(* Logix 5000 project; controller PBS_Perfusion vendor 1 type 14 code 217 rev 32.14; software revision 32.03; part 11 of 27 *)
(* tags used below, declared in another part *)
   Inp_FdbkA : BOOL;   // Input Signal: Feedback A from device
   Inp_FdbkB : BOOL;   // Input Signal: Feedback B from device
   Inp_FdbkC : BOOL;   // Input Signal: Feedback C from device
   Inp_FdbkD : BOOL;   // Input Signal: Feedback D from device
   Inp_DeviceFault : BOOL;   // Input Signal: Device Fault from device
   Inp_PermOK0 : BOOL;   // 1=Permissives OK, device can be commanded to State 0
   Inp_NBPermOK0 : BOOL;   // 1=Non-Bypassable Permissives OK, device can be commanded to State 0
   Inp_PermOK1 : BOOL;   // 1=Permissives OK, device can be commanded to State 1
   Inp_NBPermOK1 : BOOL;   // 1=Non-Bypassable Permissives OK, device can be commanded to State 1
   Inp_PermOK2 : BOOL;   // 1=Permissives OK, device can be commanded to State 2
   Inp_NBPermOK2 : BOOL;   // 1=Non-Bypassable Permissives OK, device can be commanded to State 2
   Inp_PermOK3 : BOOL;   // 1=Permissives OK, device can be commanded to State 3
   Inp_NBPermOK3 : BOOL;   // 1=Non-Bypassable Permissives OK, device can be commanded to State 3
   Inp_IntlkOK : BOOL;   // 1=Interlocks OK, 0=Not OK, go to State 0
   Inp_NBIntlkOK : BOOL;   // 1=Non-Bypassable Interlocks OK, 0=Not OK, go to State 0
   Inp_IntlkAvail : BOOL;   // 1 = Interlock Availibility OK
   Inp_IOFault : BOOL;   // Input Communication Status 0=OK, 1=fail
   Inp_Sim : BOOL;   // 1=Simulate working device; 0=Control actual device
   Inp_OvrdCmd : DINT;   // Override Device Command: 0=None, 1=St.0, 2=St.1, 3=St.2, 4=St.3
   Inp_HornInh : BOOL;   // 1 = Inhibit audible alert, 0 = Alllow audible alert
   Inp_Reset : BOOL;   // 1=Reset all fault conditions and latched Alarms
   Cfg_St0onShed : BOOL;   // 1=Go to State 0 on Shed, 0=Hold position on Shed
   Cfg_NumStates : DINT;   // Number of device states (2..4)
   Cfg_FdbkSt0Check : SINT;   // Bit=1: Check Feedback in state 0, Bit=0: don't care
   Cfg_FdbkSt0State : SINT;   // (if checking) Bit=1: Feedback is 1 in State 0, Bit=0: Feedback is 0
   Cfg_FdbkSt1Check : SINT;   // Bit=1: Check Feedback in state 1, Bit=0: don't care
   Cfg_FdbkSt1State : SINT;   // (if checking) Bit=1: Feedback is 1 in State 1, Bit=0: Feedback is 0
   Cfg_FdbkSt2Check : SINT;   // Bit=1: Check Feedback in state 2, Bit=0: don't care
   Cfg_FdbkSt2State : SINT;   // (if checking) Bit=1: Feedback is 1 in State 2, Bit=0: Feedback is 0
   Cfg_FdbkSt3Check : SINT;   // Bit=1: Check Feedback in state 3, Bit=0: don't care
   Cfg_FdbkSt3State : SINT;   // (if checking) Bit=1: Feedback is 1 in State 3, Bit=0: Feedback is 0
   Cfg_HasMoreObj : BOOL;   // 1=Tells HMI an object with more info is available
   Cfg_OperSt0Prio : BOOL;   // 1=OCmd_St0 any time, 0=OCmd_St0 only when Oper selected
   Cfg_ExtSt0Prio : BOOL;   // 1=XCmd_St0 any time, 0=XCmd_St0 only when Ext selected
   Cfg_OCmdResets : BOOL;   // 1=New device OCmd resets shed latches and cleared alarms, 0=OCmdReset req'd.
   Cfg_XCmdResets : BOOL;   // 1=New device XCmd resets shed latches and cleared alarms, 0=XCmdReset req'd.
   Cfg_OvrdPermIntlk : BOOL;   // 1=Override ignores Bypassable Perm/ Intlk; 0=always use Perm/Intlk
   Cfg_ShedOnFail : BOOL;   // 1=Go to State 0 and Alarm on Fail to reach position; 0=Alarm only on Fail
   Cfg_ShedOnDeviceFault : BOOL;   // 1=Go to State 0 and Alarm on Device Fault; 0=Alarm only on Device Fault
   Cfg_ShedOnIOFault : BOOL;   // 1=Go to State 0 and Alarm on I/O Fault; 0=Alarm only on I/O Fault
   Cfg_HornOnChange : BOOL;   // 0 = Horn on energize only, 1 = Horn on any state change
   Cfg_OutAPulseT : REAL;   // Time to pulse Output A (sec) (0=output held continuously)
   Cfg_OutBPulseT : REAL;   // Time to pulse Output B (sec) (0=output held continuously)
   Cfg_OutCPulseT : REAL;   // Time to pulse Output C (sec) (0=output held continuously)
   Cfg_OutDPulseT : REAL;   // Time to pulse Output D (sec) (0=output held continuously)
   Cfg_SimFdbkT : REAL;   // Delay to echo back reaching state when in Simulation (sec)
   Cfg_StartHornT : REAL;   // Time to sound audible on commanded start (sec) (0=disabled)
   Cfg_FailT : REAL;   // Time after new state requested to reach that state before Fault (sec)
   PSet_Owner : DINT;   // Program Owner Request ID (non-zero) or Release (zero)
   PCmd_St0 : BOOL;   // Program Command to set device to State 0
   PCmd_St1 : BOOL;   // Program Command to set device to State 1
   PCmd_St2 : BOOL;   // Program Command to set device to State 2
   PCmd_St3 : BOOL;   // Program Command to set device to State 3
   PCmd_Reset : BOOL;   // Program Command to ResetShed Latches and Cleared Alarms
   PCmd_FailAck : ALIAS FOR Fail.PCmd_Ack;   // Program Command to Acknowledge Fail to Reach Target Position Alarm
   PCmd_DeviceFaultAck : ALIAS FOR DeviceFault.PCmd_Ack;   // Program Command to Acknowledge Device Fault Alarm
   PCmd_IntlkTripAck : ALIAS FOR IntlkTrip.PCmd_Ack;   // Program Command to Acknowledge Interlock Trip Alarm
   PCmd_IOFaultAck : ALIAS FOR IOFault.PCmd_Ack;   // Program Command to Acknowledge I/O Fault Alarm
   XCmd_St0 : BOOL;   // External Command to set device to State 0
   XCmd_St1 : BOOL;   // External Command to set device to State 1
   XCmd_St2 : BOOL;   // External Command to set device to State 2
   XCmd_St3 : BOOL;   // External Command to set device to State 3
   XCmd_Reset : BOOL;   // External Command to reset shed latches and cleared alarms
   Val_Cmd : DINT;   // Device Command 0=None, 1=State 0, 2=State 1, 3=State 2, 4=State 3
   Val_Owner : DINT;   // Current Object Owner ID (0=not owned)
   Sts_Available : BOOL;   // 1=Device available for control by automation (Prog)
   Sts_Bypass : BOOL;   // 1=Bypassable Interlocks and Permissives are Bypassed
   Sts_BypActive : BOOL;   // 1=Interlock / Permissive Bypassing Active (Bypassed or Maintenance)
   Sts_NotRdy : BOOL;   // 1=Device Not Ready, see detail bits for reason
   Nrdy_CfgErr : BOOL;   // 1=Device Not Ready: Configuration Error
   Nrdy_EqpFault : BOOL;   // 1=Device Not Ready: External Equipment Fault (Fault or Shed Requires Reset)
   Nrdy_Fail : BOOL;   // 1=Device Not Ready: Device Failure (Shed Requires Reset)
   Nrdy_Intlk : BOOL;   // 1=Device Not Ready: Interlock Not OK
   Nrdy_IOFault : BOOL;   // 1=Device Not Ready: I/O Fault (Shed Requires Reset)
   Nrdy_OoS : BOOL;   // 1=Device Not Ready: Device is Out of Service
   Nrdy_PrioSt0 : BOOL;   // 1=Device Not Ready: Oper/Ext Priority State 0 Command Requires Reset
   Nrdy_Perm : BOOL;   // 1=Device Not Ready: Permissive Not OK
   Sts_MaintByp : BOOL;   // 1=Device has a Maintenance Bypass function active
   Err_Timer : BOOL;   // 1=Error in Config: Feeback Check timer preset (use 0 to 2147483)
   Err_Sim : BOOL;   // 1=Error in Config: Simulation timer preset (use 0 to 2147483)
   Sts_Hand : ALIAS FOR CmdSrc.Sts_Hand;
   Sts_OoS : ALIAS FOR CmdSrc.Sts_OoS;
   Sts_Maint : ALIAS FOR CmdSrc.Sts_Maint;
   Sts_Ovrd : ALIAS FOR CmdSrc.Sts_Ovrd;
   Sts_Ext : ALIAS FOR CmdSrc.Sts_Ext;
   Sts_Prog : ALIAS FOR CmdSrc.Sts_Prog;
   Sts_Oper : ALIAS FOR CmdSrc.Sts_Oper;
   Sts_Fail : ALIAS FOR Fail.Inp;   // 1=Device failed to reach commended state
   Sts_DeviceFault : ALIAS FOR DeviceFault.Inp;   // 1=Device Fault (from Inp_DeviceFault)
   Sts_IntlkTrip : ALIAS FOR IntlkTrip.Inp;   // 1=Device commanded to State 0 by an Interlock NOT OK (one-shot)
   Sts_IOFault : ALIAS FOR IOFault.Inp;   // I/O Comm Fault Status (0=OK, 1=Bad)
   P_D4SD : BOOL;   // Unique Parameter Name for auto - discovery
   Wrk_OutDPulseT : TIMER;   // Output D Pulse Timer
   Wrk_OutCPulseT : TIMER;   // Output C Pulse Timer
   Wrk_OutBPulseT : TIMER;   // Output B Pulse Timer
   Wrk_OutAPulseT : TIMER;   // Output A Pulse Timer
   Wrk_Bypass : BOOL;   // Internal Bypassable Permissives and Interlocks are Bypassed flag
   Wrk_ActState : DINT;   // Actual State (enum)
   Fail : P_Alarm;   // Device Fail to reach commanded position
   DeviceFault : P_Alarm;   // Device Fault from device via input
   CmdSrc : P_CmdSrc;   // Control / Command Source Selection
   IOFault : P_Alarm;   // I/O Fault Alarm
   IntlkTrip : P_Alarm;   // Interlock Trip Alarm
   Wrk_ONS : SINT;   // One-Shot Store Bits
   Wrk_FdbkState : DINT;   // State(s) of device as shown by feedbacks
   Cfg_Tag : STRING_20;   // Tagname for display on HMI
   Cfg_Label : STRING_20;   // Label for graphic symbol displayed on HMI
   Cfg_Desc : STRING_40;   // Description for display on HMI
   Cfg_St3Text : STRING_8;   // Text to display in State 3
   Cfg_St2Text : STRING_8;   // Text to display in State 2
   Cfg_St1Text : STRING_8;   // Text to display in State 1
   Cfg_St0Text : STRING_8;   // Text to display in State 0
   Wrk_PermOK3 : BOOL;   // 1=Permissives are OK to go to state 3
   Wrk_PermOK2 : BOOL;   // 1=Permissives are OK to go to state 2
   Wrk_PermOK1 : BOOL;   // 1=Permissives are OK to go to state 1
   Wrk_PermOK0 : BOOL;   // 1=Permissives are OK to go to state 0
   Wrk_TgtState : DINT;   // Target device state as a number (0, 1, 2 or 3)
   Wrk_SimT : TIMER;   // Time "moving" before going to target pos. in simulation
   Wrk_FailT : TIMER;   // Failure Check timer (time to reach target position)
   Wrk_NewCmd : BOOL;   // 1=A state command has been received (even for same state)
   Wrk_PrevTgt : DINT;   // Previous Target State (last scan)
   HMI_Type : STRING_16;   // Type identifier for HMI navigation
   HMI_Lib : STRING_12;   // Display Library for Faceplate call-up
   Wrk_NotRdy : BOOL;   // Device Not Ready conditions excluding shed latches
   Wrk_NotRdy1 : BOOL;   // Device Not Ready excluding only Permissives
   Wrk_NoLongerSim : BOOL;   // Switched from Simulated to Real Device this scan
   Cfg_Area : STRING_Area;   // Process Area for security
   MRdy_Check : BOOL;   // 1=Ready for MCmd_Check, enable HMI button
   MRdy_Bypass : BOOL;   // 1=Ready for MCmd_Bypass, enable HMI button
   OCmd_ResetAckAll : BOOL;   // Oper Cmd to reset shed latches and cleared alarms, plus Acknowledge alarms
   OCmd_Reset : BOOL;   // Oper Cmd to reset shed latches and cleared alarms
   OCmd_St3 : BOOL;   // Operator Command to set device to State 3
   OCmd_St2 : BOOL;   // Operator Command to set device to State 2
   OCmd_St1 : BOOL;   // Operator Command to set device to State 1
   OCmd_St0 : BOOL;   // Operator Command to set device to State 0
   MCmd_Check : BOOL;   // Maintenance Command to Check Interlocks and Permissives
   MCmd_Bypass : BOOL;   // Maintenance Command to Bypass Interlocks and Permissives
   Wrk_StartHornT : TIMER;   // Timer for audible alert or start
   Wrk_StartHorn : BOOL;   // 1=Sound audible prior to commanded energize/ state change
   Wrk_TgtStateTmp : DINT;   // Target device state as a number (0, 1, 2 or 3) stored, before audible alert
   Wrk_AfterHornONS : BOOL;
   Wrk_AfterHornONS2 : BOOL;
   ONS : DINT[3];
   REAL : DINT;
(* P_D4SD, continued *)

ROUTINE Logic   (* ladder *)
// Normal Scan: control / monitor 2-, 3- or 4-State device
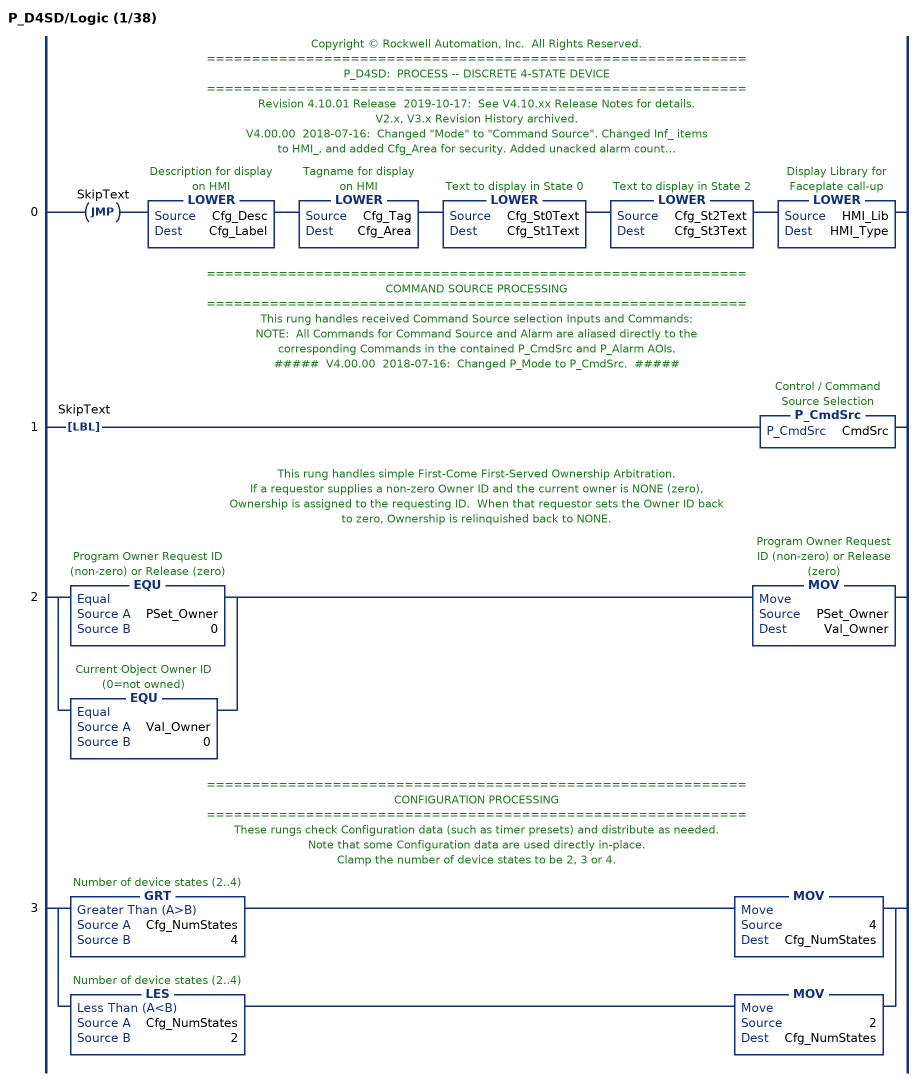
   // Copyright © Rockwell Automation, Inc.  All Rights Reserved.
   // ============================================================
   // P_D4SD:  PROCESS -- DISCRETE 4-STATE DEVICE
   // ============================================================
   // Revision 4.10.01 Release  2019-10-17:  See V4.10.xx Release Notes for details.
   // V2.x, V3.x Revision History archived.
   // V4.00.00  2018-07-16:  Changed "Mode" to "Command Source". Changed Inf_ items
   // to HMI_, and added Cfg_Area for security. Added unacked alarm count.
   // Deleted Cfg_PCmdClear; all Program Commands are now self-clearing.
   // Aligned ready bit naming with command bit names.
   // All OCmds/MCmds and ORdys/MRdys are now Local Tags.
   // Added Sts_AckReqd and Sts_ResetReqd for use by external objects.
   // Changed delay / time configuration items to REAL seconds.
   // V4.10.00  2019-03-08:  Changed availability to use input availability from interlocks.
   // Added audible alert on commanded energize/state change.
   // Added Inp_HornInh to disable Horn operation.
   // Modified logic to correct confgigurable shed action.
   // Updated to P_CmdSrc V4.10.00. Added Cfg_HasMoreObj.
   // V4.10.01  2019-10-17:  No changes, uprevved because P_CmdSrc 4.10.01 is used.
   // ============================================================
   // This Instruction controls and monitors feedback from
   // a Discrete 2-State, 3-State or 4-State Device, and provides:
   // *  Operator and Program Commands to select one of the 2, 3 or 4 states
   // *  User-configurable text labels for the states
   // *  Per-State setting, clearing or holding of four user-configurable outputs
   // *  Per-State monitoring of four feedbacks (on, off or don't care) to confirm state
   // *  Detection of failure to reach the target state (when feedbacks are used)
   // *  Monitoring of Permissive conditions to allow commanding to each state
   // *  Monitoring of Interlock conditions to return device to State 0
   // *  Simulation, providing feedback of a working device while
   //       disabling output (keeping de-energized)
   // *  Monitoring of I/O communication status
   // *  Alarms for Fail to reach target state (if feedbacks are used), Device Failure
   // (reported by device using an input), Interlock Trip, I/O Fault
   // *  "Available" status for use by automation logic to know whether
   //      the device can be controlled by other objects.
   // Command Sources are arbitrated by a P_CmdSrc Add-On Instruction instance.
   // Command Sources: Operator, Program, External, Override, Maintenance, Out of
   // Service, Hand.  Alarms are provided by P_Alarm Add-On Instruction instances.
   // ============================================================
   // SHOW LOCAL STRINGS
   // ============================================================
   // The STRINGs containing the text associated with each instance of this
   // instruction cannot be Input or Output Parameters, because STRINGs are not
   //  'atomic' types. (Inputs and Outputs must be SINT, INT, DINT, REAL, or BOOL.)
   // In order to make it easier to find and configure these STRINGs, this rung
   // was added.  THE JMP (and the LBL on the following rung)
   // MUST NOT BE REMOVED!!!
   // To view the STRINGs, go to the instruction instance (in LD or FBD), RIGHT-click
   // to bring up the context menu and select "Open Instruction Logic".
   // This rung will appear with the STRING values for the selected instance.
   // You may double-click the STRING values here to modify them as well.
   // #####  V4.00.00  2018-07-16:  Added string for Cfg_Area, renamed Inf_* to HMI_*.  #####
   0: JMP(SkipText)LOWER(Cfg_Desc,Cfg_Label)LOWER(Cfg_Tag,Cfg_Area)LOWER(Cfg_St0Text,Cfg_St1Text)LOWER(Cfg_St2Text,Cfg_St3Text)LOWER(HMI_Lib,HMI_Type);
   // ============================================================
   // COMMAND SOURCE PROCESSING
   // ============================================================
   // This rung handles received Command Source selection Inputs and Commands:
   // NOTE:  All Commands for Command Source and Alarm are aliased directly to the
   // corresponding Commands in the contained P_CmdSrc and P_Alarm AOIs.
   // #####  V4.00.00  2018-07-16:  Changed P_Mode to P_CmdSrc.  #####
   1: LBL(SkipText)P_CmdSrc(CmdSrc);
   // This rung handles simple First-Come First-Served Ownership Arbitration.
   // If a requestor supplies a non-zero Owner ID and the current owner is NONE (zero),
   // Ownership is assigned to the requesting ID.  When that requestor sets the Owner ID back
   // to zero, Ownership is relinquished back to NONE.
   2: [EQU(PSet_Owner,0) ,EQU(Val_Owner,0) ]MOV(PSet_Owner,Val_Owner);
   // ============================================================
   // CONFIGURATION PROCESSING
   // ============================================================
   // These rungs check Configuration data (such as timer presets) and distribute as needed.
   // Note that some Configuration data are used directly in-place.
   // Clamp the number of device states to be 2, 3 or 4.
   3: [GRT(Cfg_NumStates,4) MOV(4,Cfg_NumStates) ,LES(Cfg_NumStates,2) MOV(2,Cfg_NumStates) ];
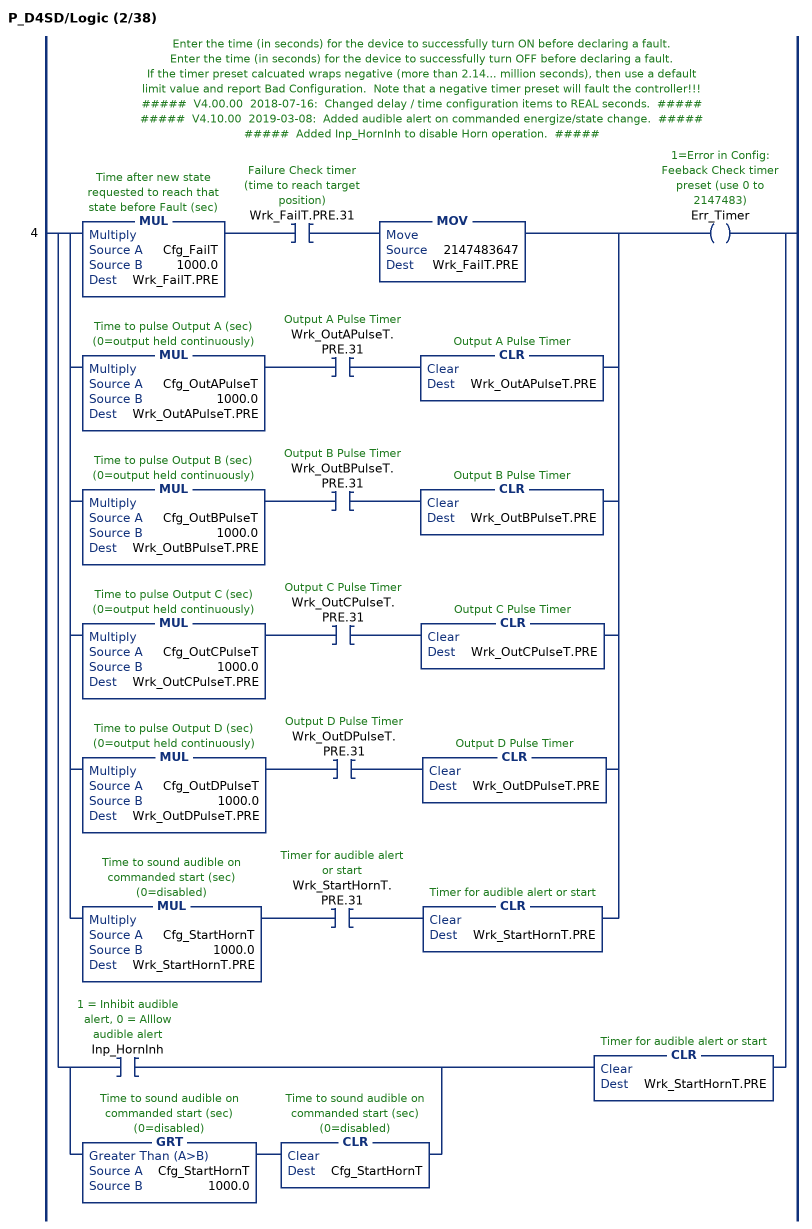
   // Enter the time (in seconds) for the device to successfully turn ON before declaring a fault.
   // Enter the time (in seconds) for the device to successfully turn OFF before declaring a fault.
   // If the timer preset calcuated wraps negative (more than 2.14... million seconds), then use a default
   // limit value and report Bad Configuration.  Note that a negative timer preset will fault the controller!!!
   // #####  V4.00.00  2018-07-16:  Changed delay / time configuration items to REAL seconds.  #####
   // #####  V4.10.00  2019-03-08:  Added audible alert on commanded energize/state change.  #####
   // #####  Added Inp_HornInh to disable Horn operation.  #####
   4: [[MUL(Cfg_FailT,1000.0,Wrk_FailT.PRE) XIC(Wrk_FailT.PRE.31) MOV(2147483647,Wrk_FailT.PRE) ,MUL(Cfg_OutAPulseT,1000.0,Wrk_OutAPulseT.PRE) XIC(Wrk_OutAPulseT.PRE.31) CLR(Wrk_OutAPulseT.PRE) ,MUL(Cfg_OutBPulseT,1000.0,Wrk_OutBPulseT.PRE) XIC(Wrk_OutBPulseT.PRE.31) CLR(Wrk_OutBPulseT.PRE) ,MUL(Cfg_OutCPulseT,1000.0,Wrk_OutCPulseT.PRE) XIC(Wrk_OutCPulseT.PRE.31) CLR(Wrk_OutCPulseT.PRE) ,MUL(Cfg_OutDPulseT,1000.0,Wrk_OutDPulseT.PRE) XIC(Wrk_OutDPulseT.PRE.31) CLR(Wrk_OutDPulseT.PRE) ,MUL(Cfg_StartHornT,1000.0,Wrk_StartHornT.PRE) XIC(Wrk_StartHornT.PRE.31) CLR(Wrk_StartHornT.PRE) ] OTE(Err_Timer) ,[XIC(Inp_HornInh) ,GRT(Cfg_StartHornT,1000.0) CLR(Cfg_StartHornT) ] CLR(Wrk_StartHornT.PRE) ];
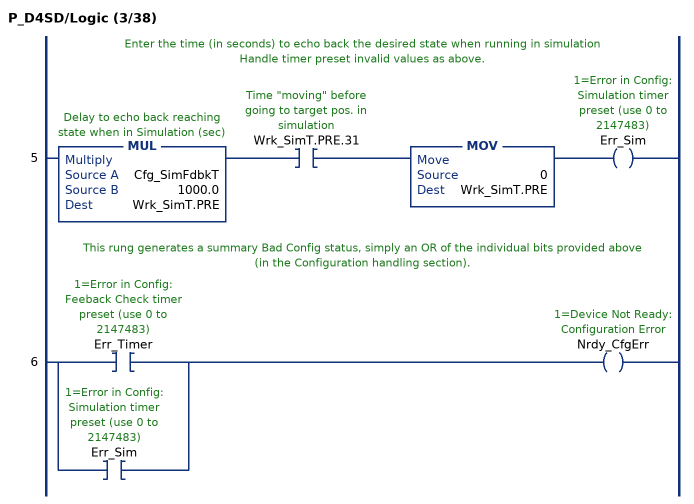
   // Enter the time (in seconds) to echo back the desired state when running in simulation
   // Handle timer preset invalid values as above.
   5: MUL(Cfg_SimFdbkT,1000.0,Wrk_SimT.PRE)XIC(Wrk_SimT.PRE.31)MOV(0,Wrk_SimT.PRE)OTE(Err_Sim);
   // This rung generates a summary Bad Config status, simply an OR of the individual bits provided above
   // (in the Configuration handling section).
   6: [XIC(Err_Timer) ,XIC(Err_Sim) ]OTE(Nrdy_CfgErr);
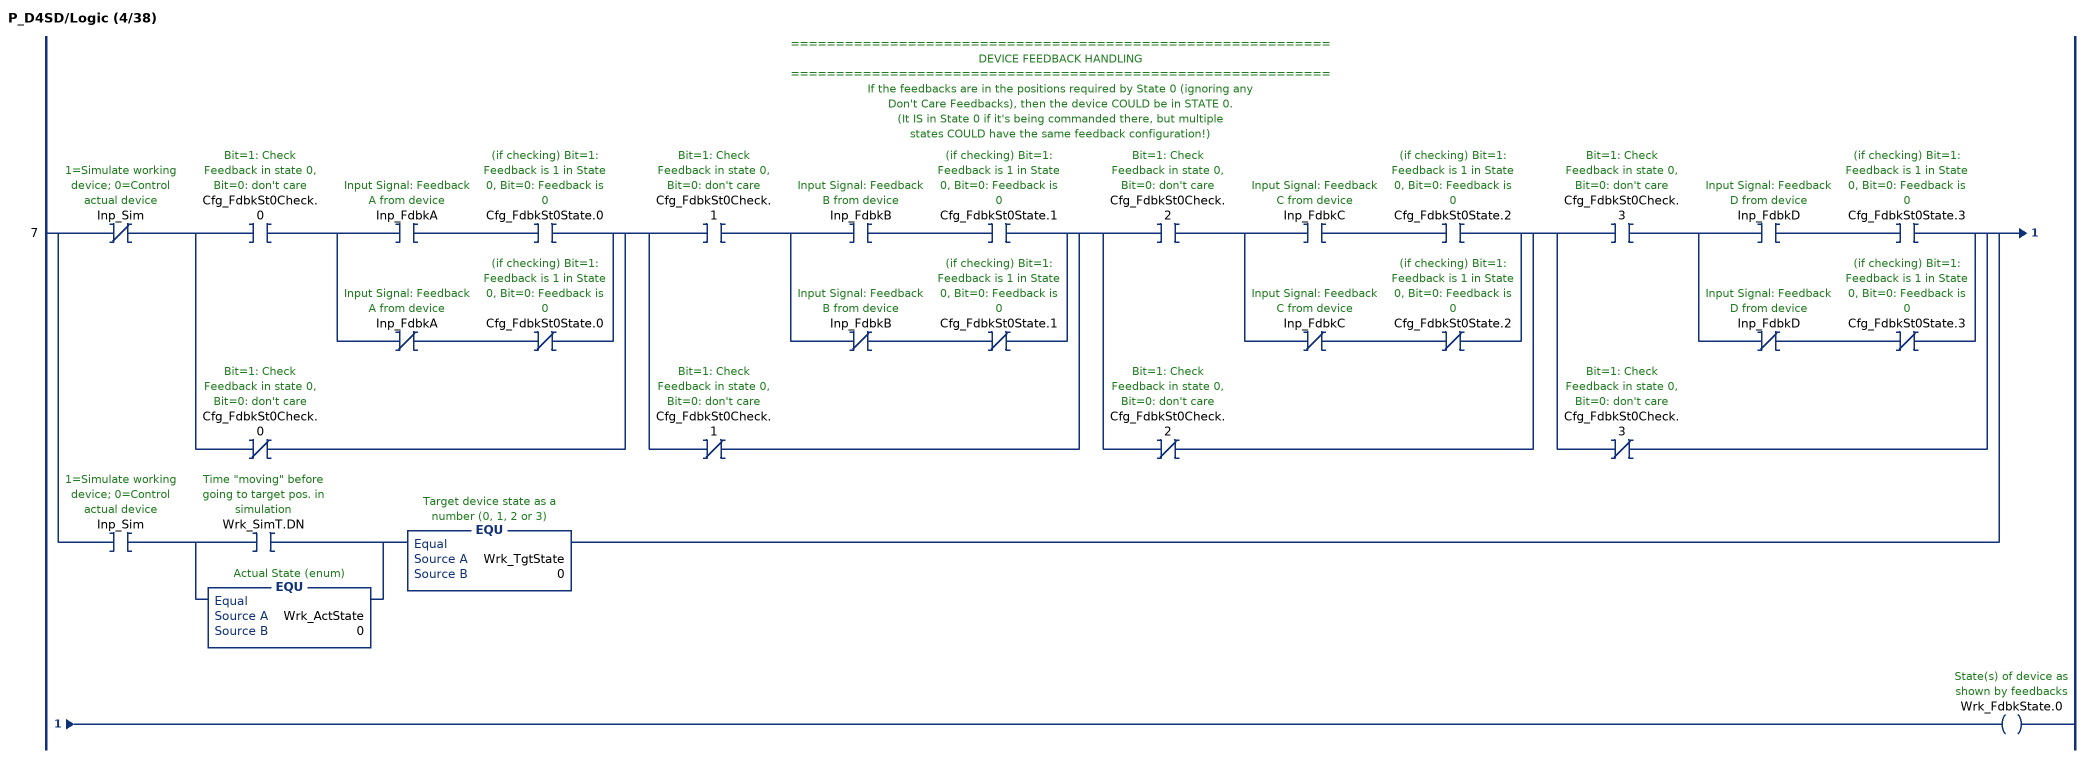
   // ============================================================
   // DEVICE FEEDBACK HANDLING
   // ============================================================
   // If the feedbacks are in the positions required by State 0 (ignoring any
   // Don't Care Feedbacks), then the device COULD be in STATE 0.
   // (It IS in State 0 if it's being commanded there, but multiple
   // states COULD have the same feedback configuration!)
   7: [XIO(Inp_Sim) [XIC(Cfg_FdbkSt0Check.0) [XIC(Inp_FdbkA) XIC(Cfg_FdbkSt0State.0) ,XIO(Inp_FdbkA) XIO(Cfg_FdbkSt0State.0) ] ,XIO(Cfg_FdbkSt0Check.0) ] [XIC(Cfg_FdbkSt0Check.1) [XIC(Inp_FdbkB) XIC(Cfg_FdbkSt0State.1) ,XIO(Inp_FdbkB) XIO(Cfg_FdbkSt0State.1) ] ,XIO(Cfg_FdbkSt0Check.1) ] [XIC(Cfg_FdbkSt0Check.2) [XIC(Inp_FdbkC) XIC(Cfg_FdbkSt0State.2) ,XIO(Inp_FdbkC) XIO(Cfg_FdbkSt0State.2) ] ,XIO(Cfg_FdbkSt0Check.2) ] [XIC(Cfg_FdbkSt0Check.3) [XIC(Inp_FdbkD) XIC(Cfg_FdbkSt0State.3) ,XIO(Inp_FdbkD) XIO(Cfg_FdbkSt0State.3) ] ,XIO(Cfg_FdbkSt0Check.3) ] ,XIC(Inp_Sim) [XIC(Wrk_SimT.DN) ,EQU(Wrk_ActState,0) ] EQU(Wrk_TgtState,0) ]OTE(Wrk_FdbkState.0);
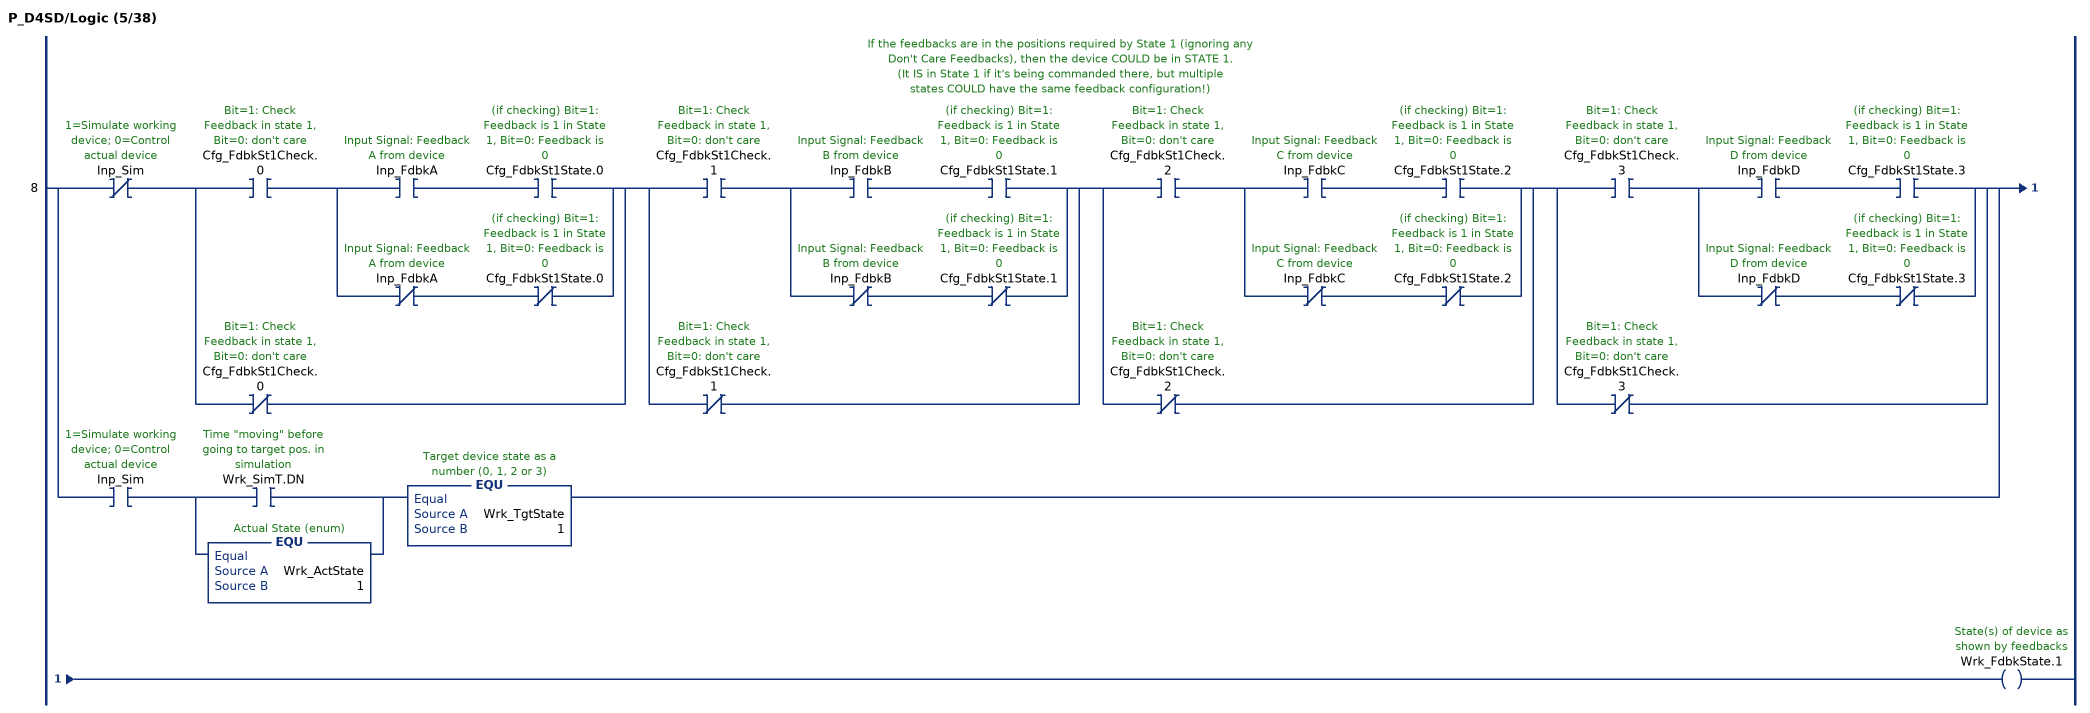
   // If the feedbacks are in the positions required by State 1 (ignoring any
   // Don't Care Feedbacks), then the device COULD be in STATE 1.
   // (It IS in State 1 if it's being commanded there, but multiple
   // states COULD have the same feedback configuration!)
   8: [XIO(Inp_Sim) [XIC(Cfg_FdbkSt1Check.0) [XIC(Inp_FdbkA) XIC(Cfg_FdbkSt1State.0) ,XIO(Inp_FdbkA) XIO(Cfg_FdbkSt1State.0) ] ,XIO(Cfg_FdbkSt1Check.0) ] [XIC(Cfg_FdbkSt1Check.1) [XIC(Inp_FdbkB) XIC(Cfg_FdbkSt1State.1) ,XIO(Inp_FdbkB) XIO(Cfg_FdbkSt1State.1) ] ,XIO(Cfg_FdbkSt1Check.1) ] [XIC(Cfg_FdbkSt1Check.2) [XIC(Inp_FdbkC) XIC(Cfg_FdbkSt1State.2) ,XIO(Inp_FdbkC) XIO(Cfg_FdbkSt1State.2) ] ,XIO(Cfg_FdbkSt1Check.2) ] [XIC(Cfg_FdbkSt1Check.3) [XIC(Inp_FdbkD) XIC(Cfg_FdbkSt1State.3) ,XIO(Inp_FdbkD) XIO(Cfg_FdbkSt1State.3) ] ,XIO(Cfg_FdbkSt1Check.3) ] ,XIC(Inp_Sim) [XIC(Wrk_SimT.DN) ,EQU(Wrk_ActState,1) ] EQU(Wrk_TgtState,1) ]OTE(Wrk_FdbkState.1);
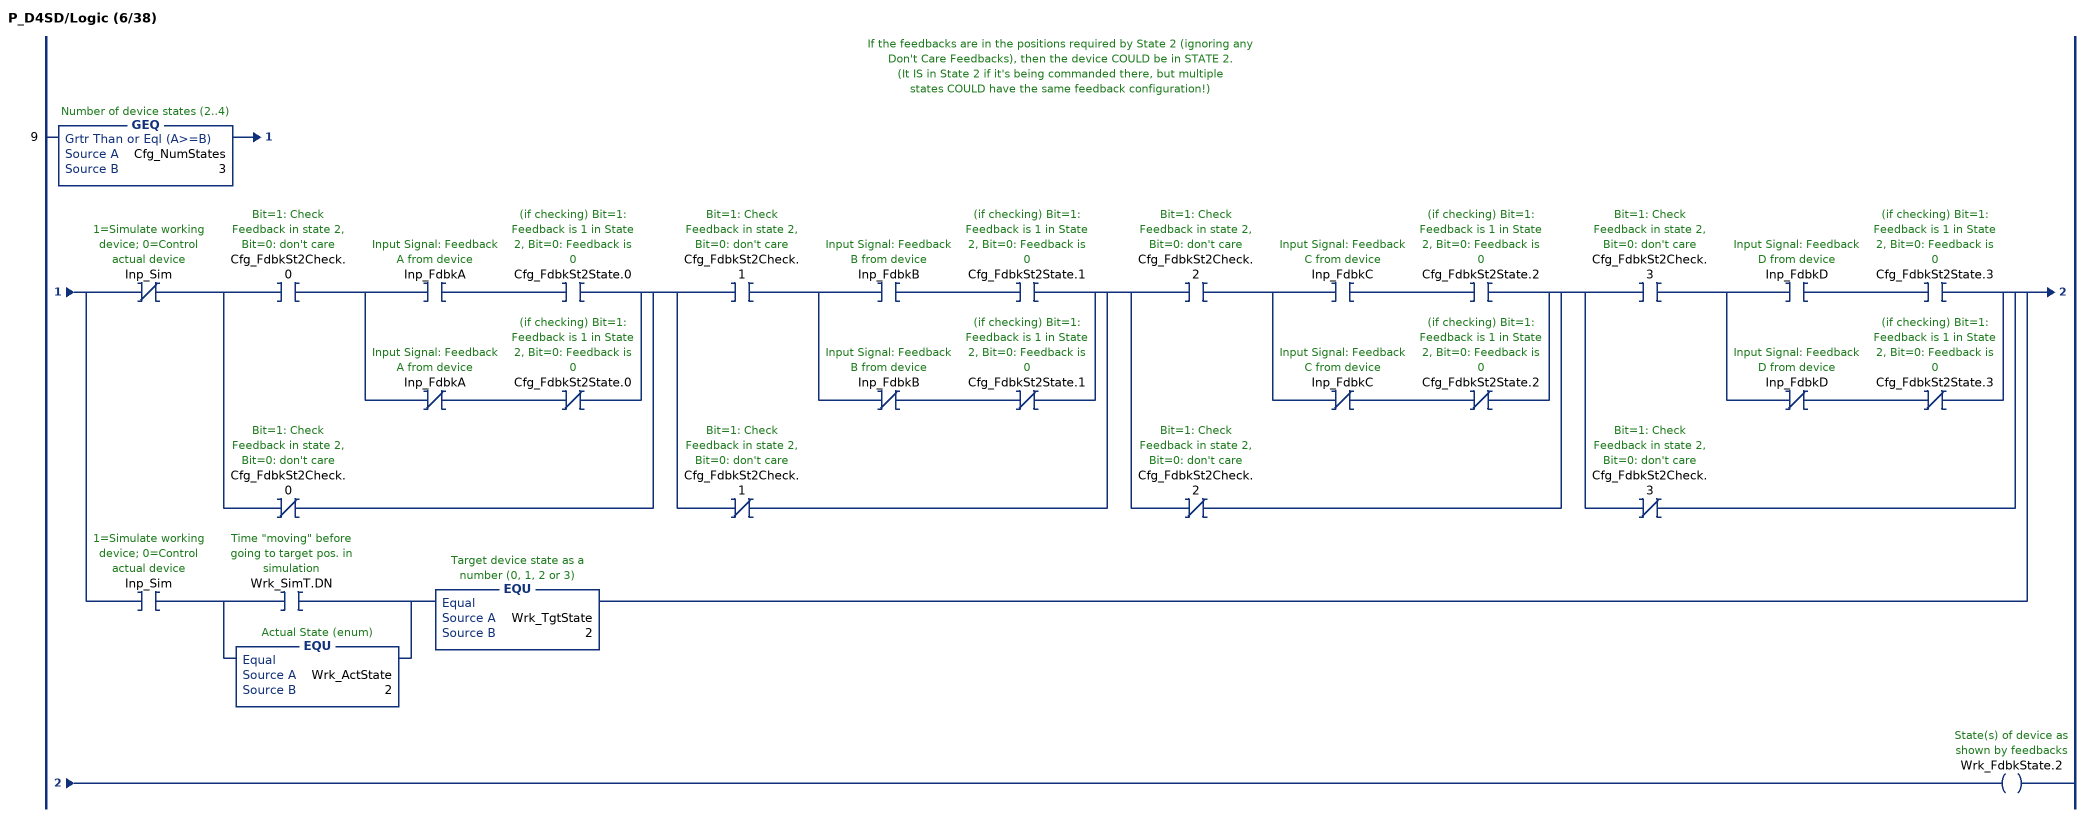
   // If the feedbacks are in the positions required by State 2 (ignoring any
   // Don't Care Feedbacks), then the device COULD be in STATE 2.
   // (It IS in State 2 if it's being commanded there, but multiple
   // states COULD have the same feedback configuration!)
   9: GEQ(Cfg_NumStates,3)[XIO(Inp_Sim) [XIC(Cfg_FdbkSt2Check.0) [XIC(Inp_FdbkA) XIC(Cfg_FdbkSt2State.0) ,XIO(Inp_FdbkA) XIO(Cfg_FdbkSt2State.0) ] ,XIO(Cfg_FdbkSt2Check.0) ] [XIC(Cfg_FdbkSt2Check.1) [XIC(Inp_FdbkB) XIC(Cfg_FdbkSt2State.1) ,XIO(Inp_FdbkB) XIO(Cfg_FdbkSt2State.1) ] ,XIO(Cfg_FdbkSt2Check.1) ] [XIC(Cfg_FdbkSt2Check.2) [XIC(Inp_FdbkC) XIC(Cfg_FdbkSt2State.2) ,XIO(Inp_FdbkC) XIO(Cfg_FdbkSt2State.2) ] ,XIO(Cfg_FdbkSt2Check.2) ] [XIC(Cfg_FdbkSt2Check.3) [XIC(Inp_FdbkD) XIC(Cfg_FdbkSt2State.3) ,XIO(Inp_FdbkD) XIO(Cfg_FdbkSt2State.3) ] ,XIO(Cfg_FdbkSt2Check.3) ] ,XIC(Inp_Sim) [XIC(Wrk_SimT.DN) ,EQU(Wrk_ActState,2) ] EQU(Wrk_TgtState,2) ]OTE(Wrk_FdbkState.2);
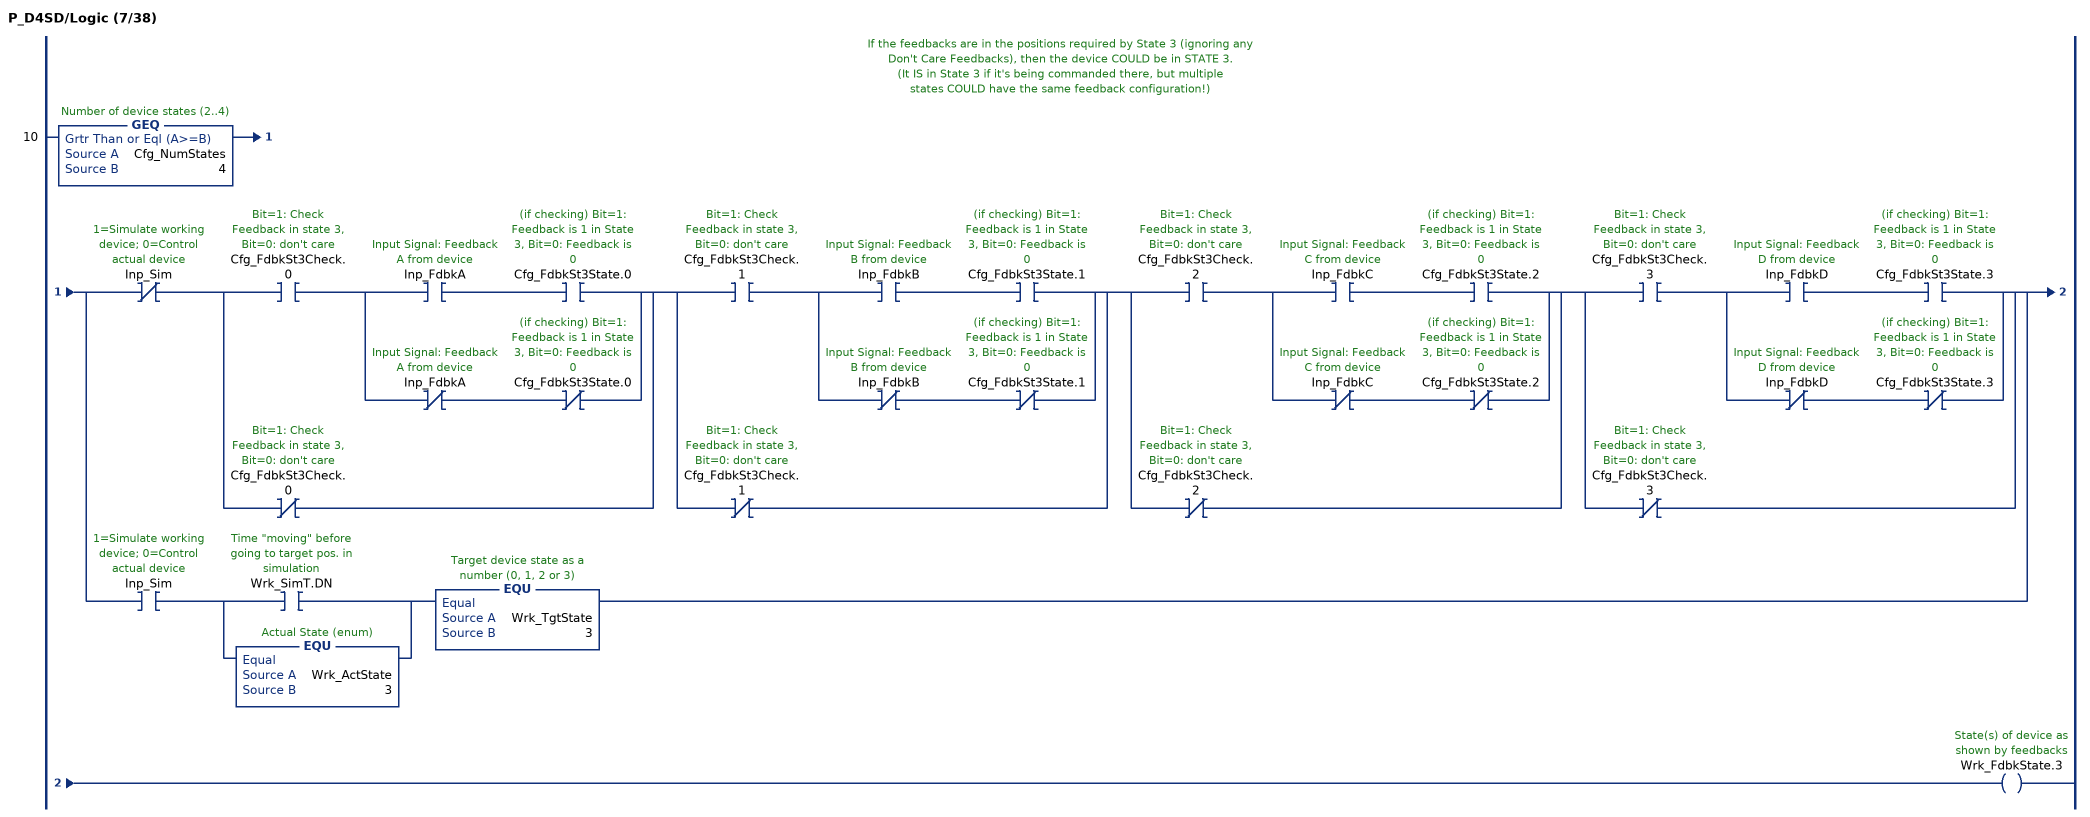
   // If the feedbacks are in the positions required by State 3 (ignoring any
   // Don't Care Feedbacks), then the device COULD be in STATE 3.
   // (It IS in State 3 if it's being commanded there, but multiple
   // states COULD have the same feedback configuration!)
   10: GEQ(Cfg_NumStates,4)[XIO(Inp_Sim) [XIC(Cfg_FdbkSt3Check.0) [XIC(Inp_FdbkA) XIC(Cfg_FdbkSt3State.0) ,XIO(Inp_FdbkA) XIO(Cfg_FdbkSt3State.0) ] ,XIO(Cfg_FdbkSt3Check.0) ] [XIC(Cfg_FdbkSt3Check.1) [XIC(Inp_FdbkB) XIC(Cfg_FdbkSt3State.1) ,XIO(Inp_FdbkB) XIO(Cfg_FdbkSt3State.1) ] ,XIO(Cfg_FdbkSt3Check.1) ] [XIC(Cfg_FdbkSt3Check.2) [XIC(Inp_FdbkC) XIC(Cfg_FdbkSt3State.2) ,XIO(Inp_FdbkC) XIO(Cfg_FdbkSt3State.2) ] ,XIO(Cfg_FdbkSt3Check.2) ] [XIC(Cfg_FdbkSt3Check.3) [XIC(Inp_FdbkD) XIC(Cfg_FdbkSt3State.3) ,XIO(Inp_FdbkD) XIO(Cfg_FdbkSt3State.3) ] ,XIO(Cfg_FdbkSt3Check.3) ] ,XIC(Inp_Sim) [XIC(Wrk_SimT.DN) ,EQU(Wrk_ActState,3) ] EQU(Wrk_TgtState,3) ]OTE(Wrk_FdbkState.3);
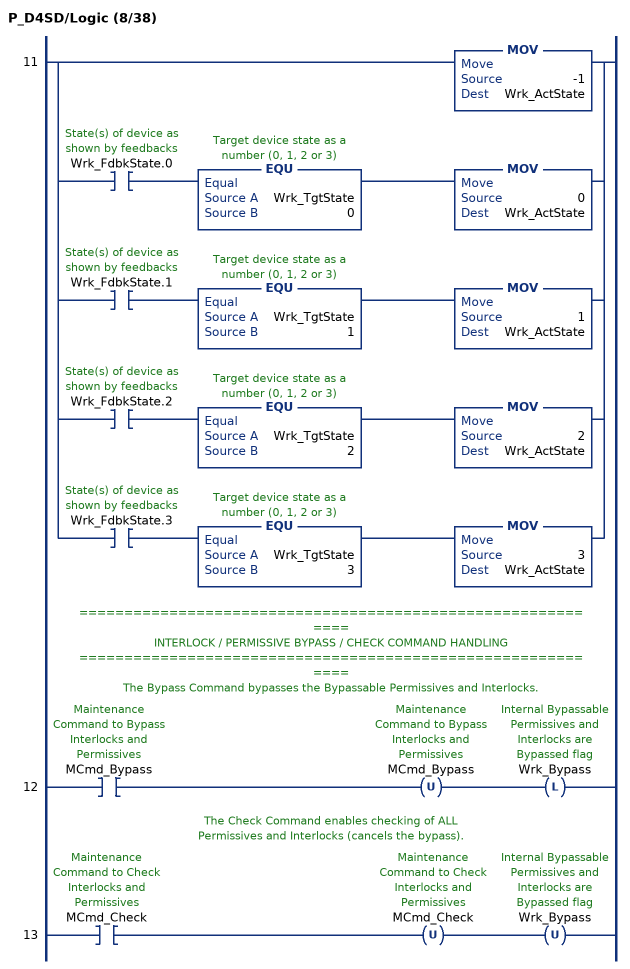
   11: [MOV(-1,Wrk_ActState) ,XIC(Wrk_FdbkState.0) EQU(Wrk_TgtState,0) MOV(0,Wrk_ActState) ,XIC(Wrk_FdbkState.1) EQU(Wrk_TgtState,1) MOV(1,Wrk_ActState) ,XIC(Wrk_FdbkState.2) EQU(Wrk_TgtState,2) MOV(2,Wrk_ActState) ,XIC(Wrk_FdbkState.3) EQU(Wrk_TgtState,3) MOV(3,Wrk_ActState) ];
   // ============================================================
   // INTERLOCK / PERMISSIVE BYPASS / CHECK COMMAND HANDLING
   // ============================================================
   // The Bypass Command bypasses the Bypassable Permissives and Interlocks.
   12: XIC(MCmd_Bypass)OTU(MCmd_Bypass)OTL(Wrk_Bypass);
   // The Check Command enables checking of ALL
   // Permissives and Interlocks (cancels the bypass).
   13: XIC(MCmd_Check)OTU(MCmd_Check)OTU(Wrk_Bypass);
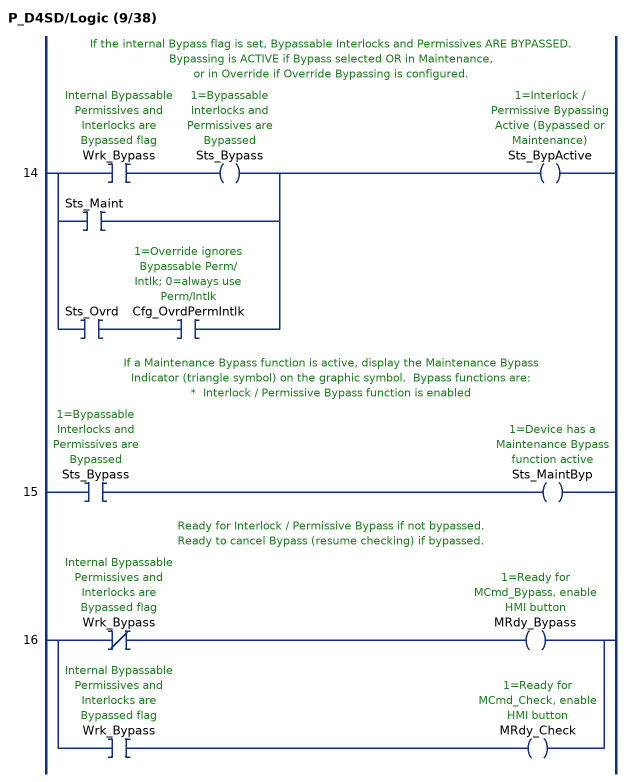
   // If the internal Bypass flag is set, Bypassable Interlocks and Permissives ARE BYPASSED.
   // Bypassing is ACTIVE if Bypass selected OR in Maintenance,
   // or in Override if Override Bypassing is configured.
   14: [XIC(Wrk_Bypass) OTE(Sts_Bypass) ,XIC(Sts_Maint) ,XIC(Sts_Ovrd) XIC(Cfg_OvrdPermIntlk) ]OTE(Sts_BypActive);
   // If a Maintenance Bypass function is active, display the Maintenance Bypass
   // Indicator (triangle symbol) on the graphic symbol.  Bypass functions are:
   // *  Interlock / Permissive Bypass function is enabled
   15: XIC(Sts_Bypass)OTE(Sts_MaintByp);
   // Ready for Interlock / Permissive Bypass if not bypassed.
   // Ready to cancel Bypass (resume checking) if bypassed.
   16: [XIO(Wrk_Bypass) OTE(MRdy_Bypass) ,XIC(Wrk_Bypass) OTE(MRdy_Check) ];
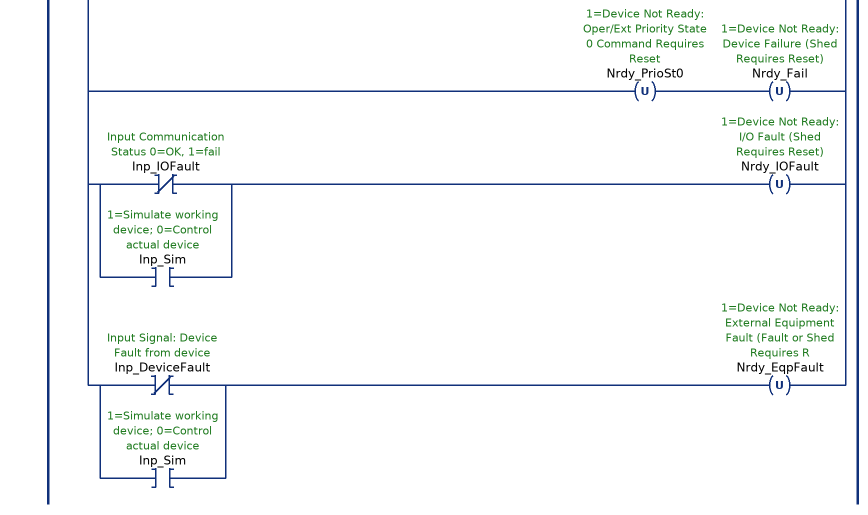
   // ============================================================
   // ALARM RESET COMMAND HANDLING
   // ============================================================
   // This rung handles the Alarm Reset Input and Commands
   // and the "Reset and Ack All" Operator Command.
   // This rung processes received Reset Commands from:
   // 1.  The Operator via HMI Operator Command, or
   // 2.  Higher-level strategies via Program Command
   // 3.  Pushbuttons or other block via Input
   // 4.  Resets initiated by other device Operator Commands (if configured to do so)
   // and forwards the Reset to ALL Alarms and latched Shed conditions.
   // #####  V4.00.00  2018-07-16:  Deleted Cfg_PCmdClear; all Program Commands are now self-clearing.  #####
   // #####  Added External Command Source and Commands.  #####
   17: [XIC(OCmd_Reset) OTU(OCmd_Reset) ,XIC(XCmd_Reset) OTU(XCmd_Reset) ,XIC(PCmd_Reset) OTU(PCmd_Reset) ,XIC(Inp_Reset) ,[XIC(OCmd_St0) XIC(Wrk_PermOK0) ,XIC(OCmd_St1) XIC(Wrk_PermOK1) ,GEQ(Cfg_NumStates,3) XIC(OCmd_St2) XIC(Wrk_PermOK2) ,GEQ(Cfg_NumStates,4) XIC(OCmd_St3) XIC(Wrk_PermOK3) ] XIC(Cfg_OCmdResets) [XIC(Sts_Oper) ,XIC(Sts_Maint) ] ,[XIC(XCmd_St0) XIC(Wrk_PermOK0) ,XIC(XCmd_St1) XIC(Wrk_PermOK1) ,GEQ(Cfg_NumStates,3) XIC(XCmd_St2) XIC(Wrk_PermOK2) ,GEQ(Cfg_NumStates,4) XIC(XCmd_St3) XIC(Wrk_PermOK3) ] XIC(Cfg_XCmdResets) XIC(Sts_Ext) ,XIC(OCmd_ResetAckAll) OTU(OCmd_ResetAckAll) [OTL(PCmd_FailAck) ,OTL(PCmd_DeviceFaultAck) ,OTL(PCmd_IntlkTripAck) ,OTL(PCmd_IOFaultAck) ] ][OTL(Fail.PCmd_Reset) OTL(DeviceFault.PCmd_Reset) ,OTL(IntlkTrip.PCmd_Reset) OTL(IOFault.PCmd_Reset) ,XIC(Sts_Fail) RES(Wrk_FailT) ,OTU(Nrdy_PrioSt0) OTU(Nrdy_Fail) ,[XIO(Inp_IOFault) ,XIC(Inp_Sim) ] OTU(Nrdy_IOFault) ,[XIO(Inp_DeviceFault) ,XIC(Inp_Sim) ] OTU(Nrdy_EqpFault) ];
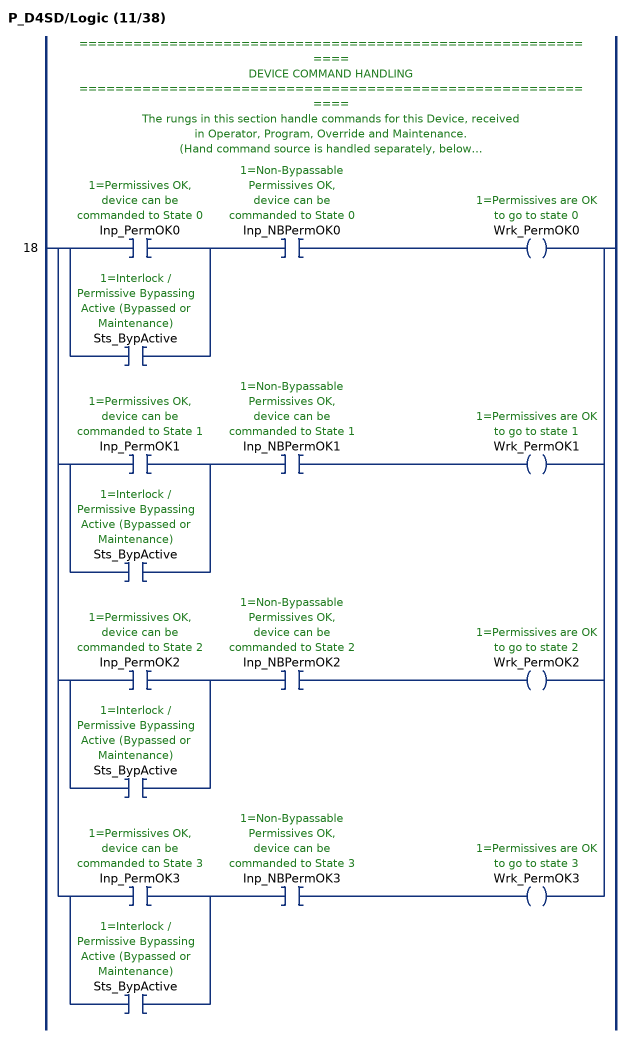
   // ============================================================
   // DEVICE COMMAND HANDLING
   // ============================================================
   // The rungs in this section handle commands for this Device, received
   // in Operator, Program, Override and Maintenance.
   // (Hand command source is handled separately, below.
   // For a command to any state, permissives for that state must be OK.
   18: [[XIC(Inp_PermOK0) ,XIC(Sts_BypActive) ] XIC(Inp_NBPermOK0) OTE(Wrk_PermOK0) ,[XIC(Inp_PermOK1) ,XIC(Sts_BypActive) ] XIC(Inp_NBPermOK1) OTE(Wrk_PermOK1) ,[XIC(Inp_PermOK2) ,XIC(Sts_BypActive) ] XIC(Inp_NBPermOK2) OTE(Wrk_PermOK2) ,[XIC(Inp_PermOK3) ,XIC(Sts_BypActive) ] XIC(Inp_NBPermOK3) OTE(Wrk_PermOK3) ];
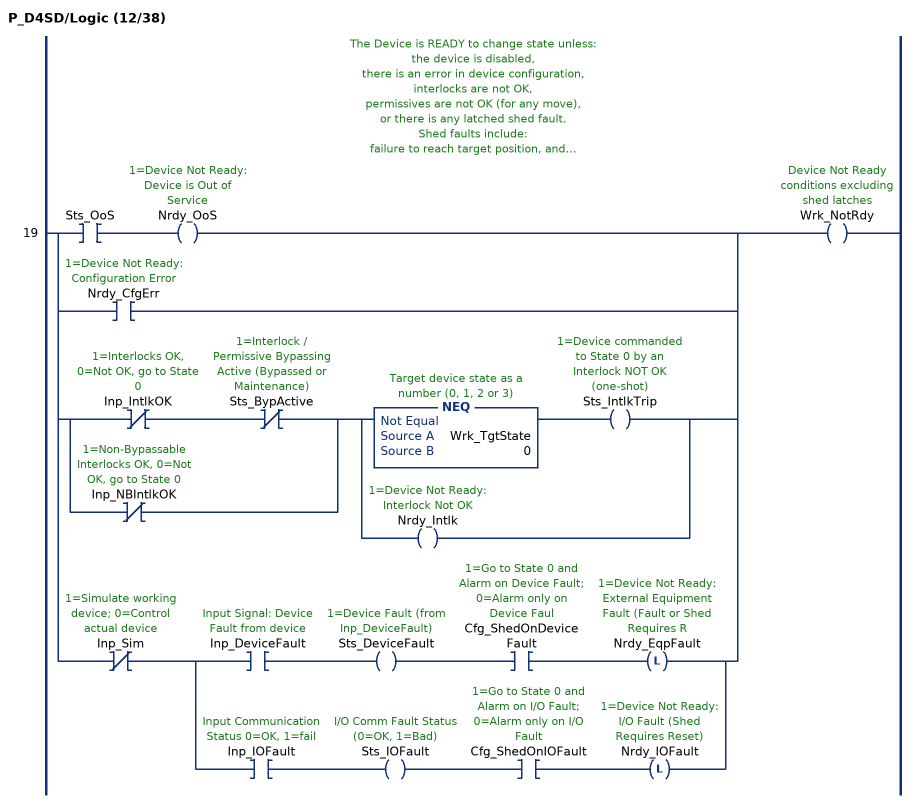
   // The Device is READY to change state unless:
   // the device is disabled,
   // there is an error in device configuration,
   // interlocks are not OK,
   // permissives are not OK (for any move),
   // or there is any latched shed fault.
   // Shed faults include:
   // failure to reach target position, and,
   // if not in simulation, a device-reported fault or I/O fault.
   // #####  V4.00.00  2018-07-16:  Disable/Enable replaced by P_CmdSrc Out of Service (OoS).  #####
   19: [XIC(Sts_OoS) OTE(Nrdy_OoS) ,XIC(Nrdy_CfgErr) ,[XIO(Inp_IntlkOK) XIO(Sts_BypActive) ,XIO(Inp_NBIntlkOK) ] [NEQ(Wrk_TgtState,0) OTE(Sts_IntlkTrip) ,OTE(Nrdy_Intlk) ] ,XIO(Inp_Sim) [XIC(Inp_DeviceFault) OTE(Sts_DeviceFault) XIC(Cfg_ShedOnDeviceFault) OTL(Nrdy_EqpFault) ,XIC(Inp_IOFault) OTE(Sts_IOFault) XIC(Cfg_ShedOnIOFault) OTL(Nrdy_IOFault) ] ]OTE(Wrk_NotRdy);
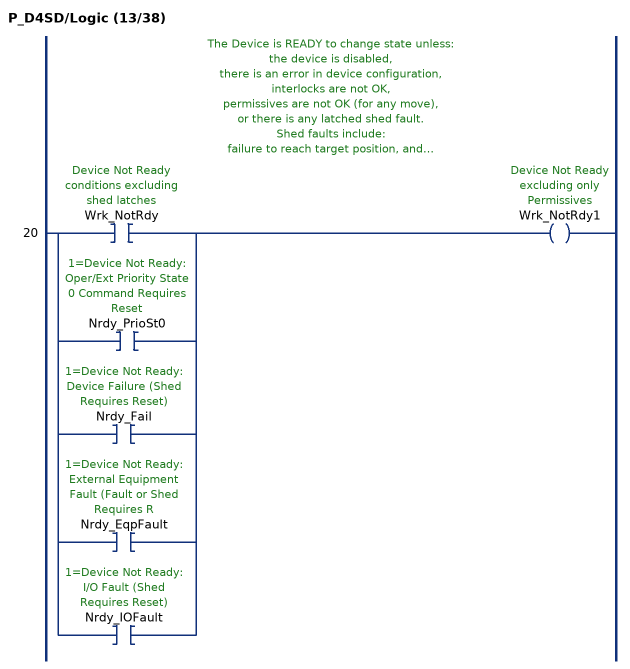
   // The Device is READY to change state unless:
   // the device is disabled,
   // there is an error in device configuration,
   // interlocks are not OK,
   // permissives are not OK (for any move),
   // or there is any latched shed fault.
   // Shed faults include:
   // failure to reach target position, and,
   // if not in simulation, a device-reported fault or I/O fault.
   20: [XIC(Wrk_NotRdy) ,XIC(Nrdy_PrioSt0) ,XIC(Nrdy_Fail) ,XIC(Nrdy_EqpFault) ,XIC(Nrdy_IOFault) ]OTE(Wrk_NotRdy1);
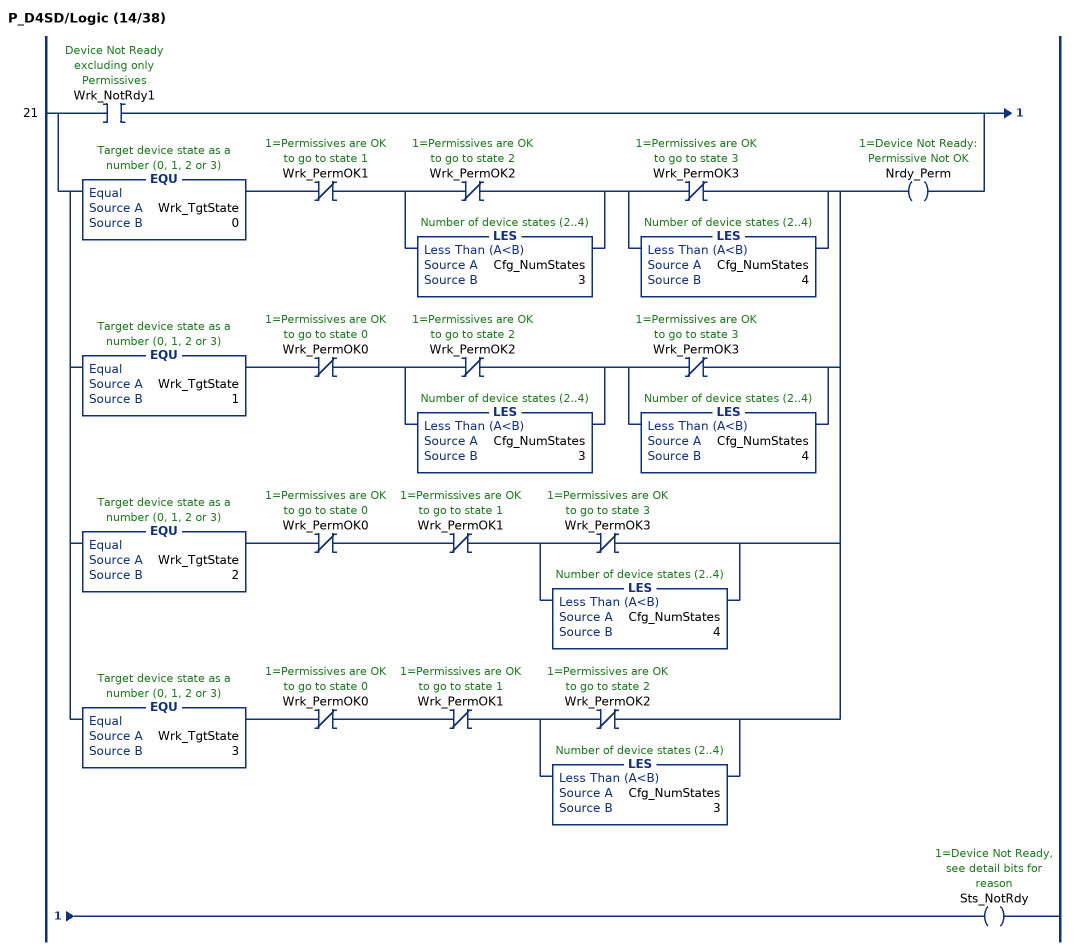
   21: [XIC(Wrk_NotRdy1) ,[EQU(Wrk_TgtState,0) XIO(Wrk_PermOK1) [XIO(Wrk_PermOK2) ,LES(Cfg_NumStates,3) ] [XIO(Wrk_PermOK3) ,LES(Cfg_NumStates,4) ] ,EQU(Wrk_TgtState,1) XIO(Wrk_PermOK0) [XIO(Wrk_PermOK2) ,LES(Cfg_NumStates,3) ] [XIO(Wrk_PermOK3) ,LES(Cfg_NumStates,4) ] ,EQU(Wrk_TgtState,2) XIO(Wrk_PermOK0) XIO(Wrk_PermOK1) [XIO(Wrk_PermOK3) ,LES(Cfg_NumStates,4) ] ,EQU(Wrk_TgtState,3) XIO(Wrk_PermOK0) XIO(Wrk_PermOK1) [XIO(Wrk_PermOK2) ,LES(Cfg_NumStates,3) ] ] OTE(Nrdy_Perm) ]OTE(Sts_NotRdy);
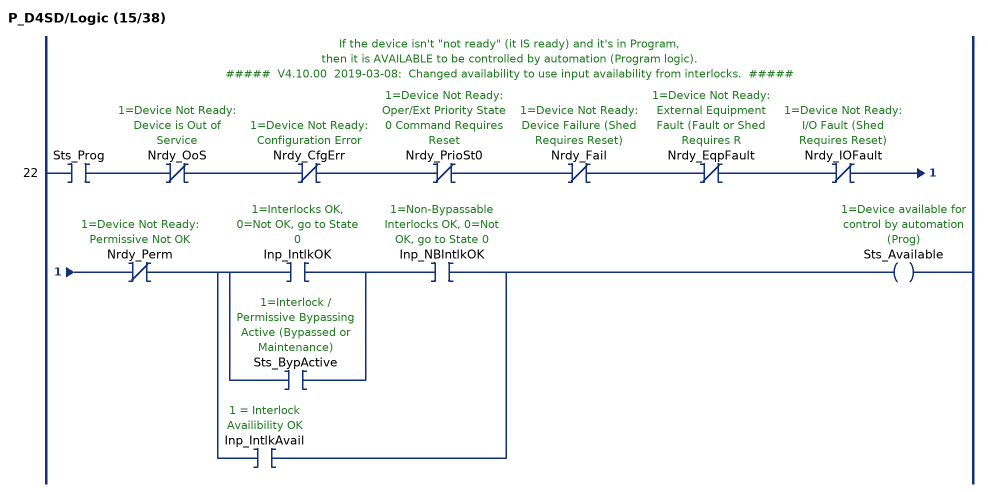
   // If the device isn't "not ready" (it IS ready) and it's in Program,
   // then it is AVAILABLE to be controlled by automation (Program logic).
   // #####  V4.10.00  2019-03-08:  Changed availability to use input availability from interlocks.  #####
   22: XIC(Sts_Prog)XIO(Nrdy_OoS)XIO(Nrdy_CfgErr)XIO(Nrdy_PrioSt0)XIO(Nrdy_Fail)XIO(Nrdy_EqpFault)XIO(Nrdy_IOFault)XIO(Nrdy_Perm)[[XIC(Inp_IntlkOK) ,XIC(Sts_BypActive) ] XIC(Inp_NBIntlkOK) ,XIC(Inp_IntlkAvail) ]OTE(Sts_Available);
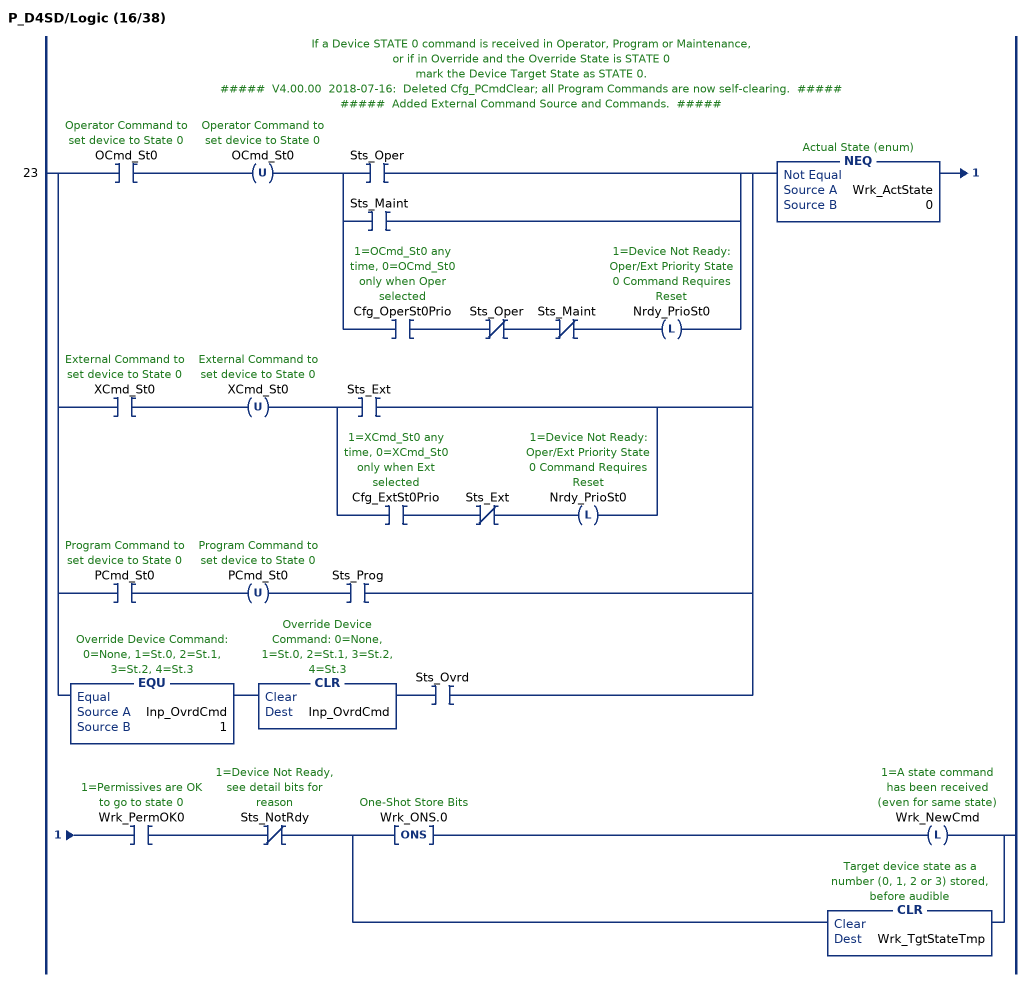
   // If a Device STATE 0 command is received in Operator, Program or Maintenance,
   // or if in Override and the Override State is STATE 0
   // mark the Device Target State as STATE 0.
   // #####  V4.00.00  2018-07-16:  Deleted Cfg_PCmdClear; all Program Commands are now self-clearing.  #####
   // #####  Added External Command Source and Commands.  #####
   23: [XIC(OCmd_St0) OTU(OCmd_St0) [XIC(Sts_Oper) ,XIC(Sts_Maint) ,XIC(Cfg_OperSt0Prio) XIO(Sts_Oper) XIO(Sts_Maint) OTL(Nrdy_PrioSt0) ] ,XIC(XCmd_St0) OTU(XCmd_St0) [XIC(Sts_Ext) ,XIC(Cfg_ExtSt0Prio) XIO(Sts_Ext) OTL(Nrdy_PrioSt0) ] ,XIC(PCmd_St0) OTU(PCmd_St0) XIC(Sts_Prog) ,EQU(Inp_OvrdCmd,1) CLR(Inp_OvrdCmd) XIC(Sts_Ovrd) ]NEQ(Wrk_ActState,0)XIC(Wrk_PermOK0)XIO(Sts_NotRdy)[ONS(Wrk_ONS.0) OTL(Wrk_NewCmd) ,CLR(Wrk_TgtStateTmp) ];
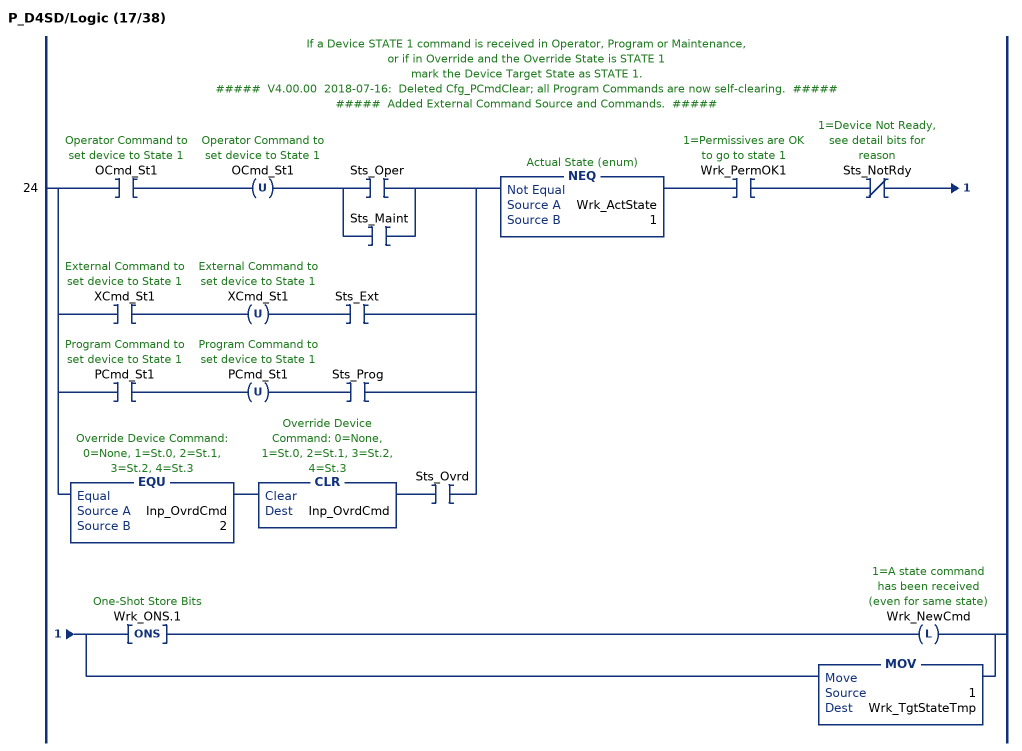
   // If a Device STATE 1 command is received in Operator, Program or Maintenance,
   // or if in Override and the Override State is STATE 1
   // mark the Device Target State as STATE 1.
   // #####  V4.00.00  2018-07-16:  Deleted Cfg_PCmdClear; all Program Commands are now self-clearing.  #####
   // #####  Added External Command Source and Commands.  #####
   24: [XIC(OCmd_St1) OTU(OCmd_St1) [XIC(Sts_Oper) ,XIC(Sts_Maint) ] ,XIC(XCmd_St1) OTU(XCmd_St1) XIC(Sts_Ext) ,XIC(PCmd_St1) OTU(PCmd_St1) XIC(Sts_Prog) ,EQU(Inp_OvrdCmd,2) CLR(Inp_OvrdCmd) XIC(Sts_Ovrd) ]NEQ(Wrk_ActState,1)XIC(Wrk_PermOK1)XIO(Sts_NotRdy)[ONS(Wrk_ONS.1) OTL(Wrk_NewCmd) ,MOV(1,Wrk_TgtStateTmp) ];
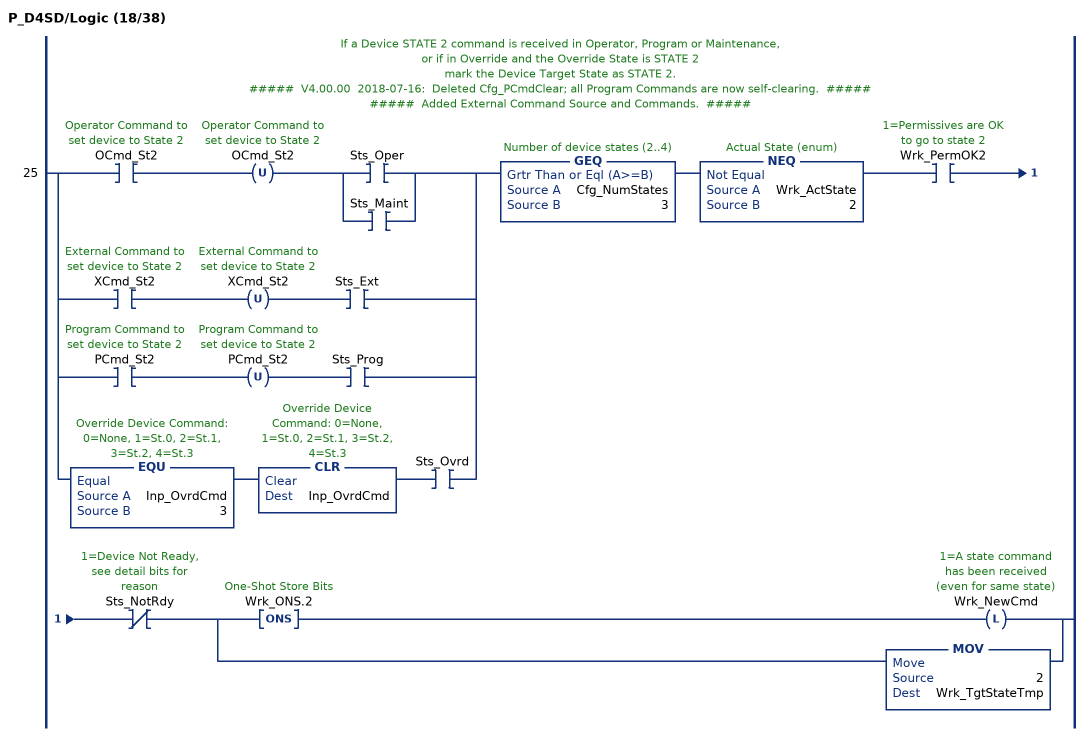
   // If a Device STATE 2 command is received in Operator, Program or Maintenance,
   // or if in Override and the Override State is STATE 2
   // mark the Device Target State as STATE 2.
   // #####  V4.00.00  2018-07-16:  Deleted Cfg_PCmdClear; all Program Commands are now self-clearing.  #####
   // #####  Added External Command Source and Commands.  #####
   25: [XIC(OCmd_St2) OTU(OCmd_St2) [XIC(Sts_Oper) ,XIC(Sts_Maint) ] ,XIC(XCmd_St2) OTU(XCmd_St2) XIC(Sts_Ext) ,XIC(PCmd_St2) OTU(PCmd_St2) XIC(Sts_Prog) ,EQU(Inp_OvrdCmd,3) CLR(Inp_OvrdCmd) XIC(Sts_Ovrd) ]GEQ(Cfg_NumStates,3)NEQ(Wrk_ActState,2)XIC(Wrk_PermOK2)XIO(Sts_NotRdy)[ONS(Wrk_ONS.2) OTL(Wrk_NewCmd) ,MOV(2,Wrk_TgtStateTmp) ];
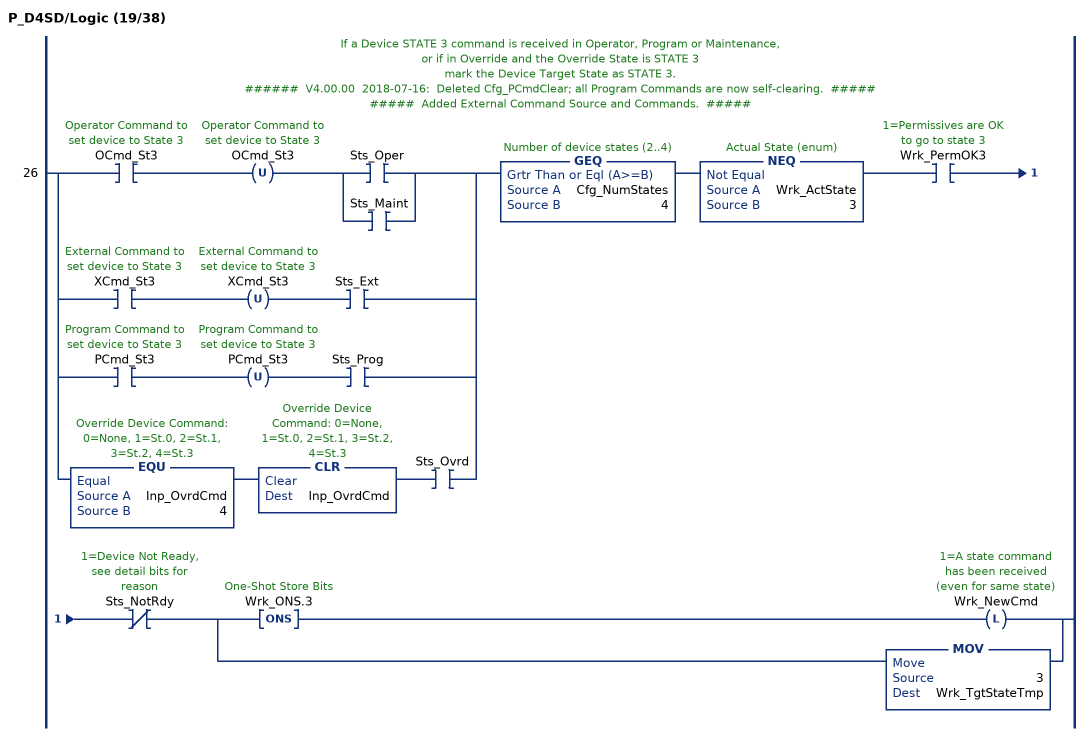
   // If a Device STATE 3 command is received in Operator, Program or Maintenance,
   // or if in Override and the Override State is STATE 3
   // mark the Device Target State as STATE 3.
   // ######  V4.00.00  2018-07-16:  Deleted Cfg_PCmdClear; all Program Commands are now self-clearing.  #####
   // #####  Added External Command Source and Commands.  #####
   26: [XIC(OCmd_St3) OTU(OCmd_St3) [XIC(Sts_Oper) ,XIC(Sts_Maint) ] ,XIC(XCmd_St3) OTU(XCmd_St3) XIC(Sts_Ext) ,XIC(PCmd_St3) OTU(PCmd_St3) XIC(Sts_Prog) ,EQU(Inp_OvrdCmd,4) CLR(Inp_OvrdCmd) XIC(Sts_Ovrd) ]GEQ(Cfg_NumStates,4)NEQ(Wrk_ActState,3)XIC(Wrk_PermOK3)XIO(Sts_NotRdy)[ONS(Wrk_ONS.3) OTL(Wrk_NewCmd) ,MOV(3,Wrk_TgtStateTmp) ];
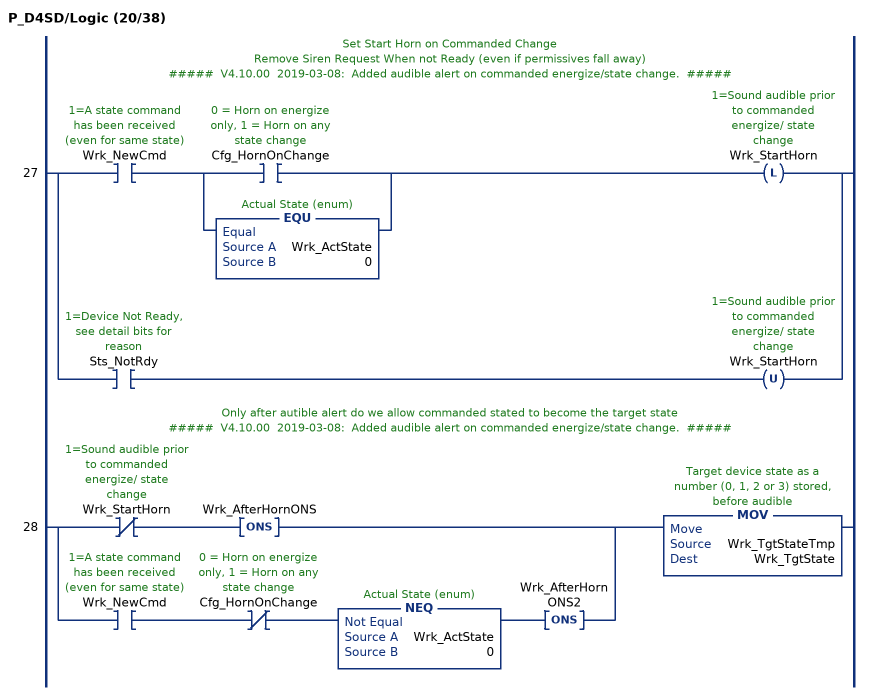
   // Set Start Horn on Commanded Change
   // Remove Siren Request When not Ready (even if permissives fall away)
   // #####  V4.10.00  2019-03-08:  Added audible alert on commanded energize/state change.  #####
   27: [XIC(Wrk_NewCmd) [XIC(Cfg_HornOnChange) ,EQU(Wrk_ActState,0) ] OTL(Wrk_StartHorn) ,XIC(Sts_NotRdy) OTU(Wrk_StartHorn) ];
   // Only after autible alert do we allow commanded stated to become the target state
   // #####  V4.10.00  2019-03-08:  Added audible alert on commanded energize/state change.  #####
   28: [XIO(Wrk_StartHorn) ONS(Wrk_AfterHornONS) ,XIC(Wrk_NewCmd) XIO(Cfg_HornOnChange) NEQ(Wrk_ActState,0) ONS(Wrk_AfterHornONS2) ]MOV(Wrk_TgtStateTmp,Wrk_TgtState);
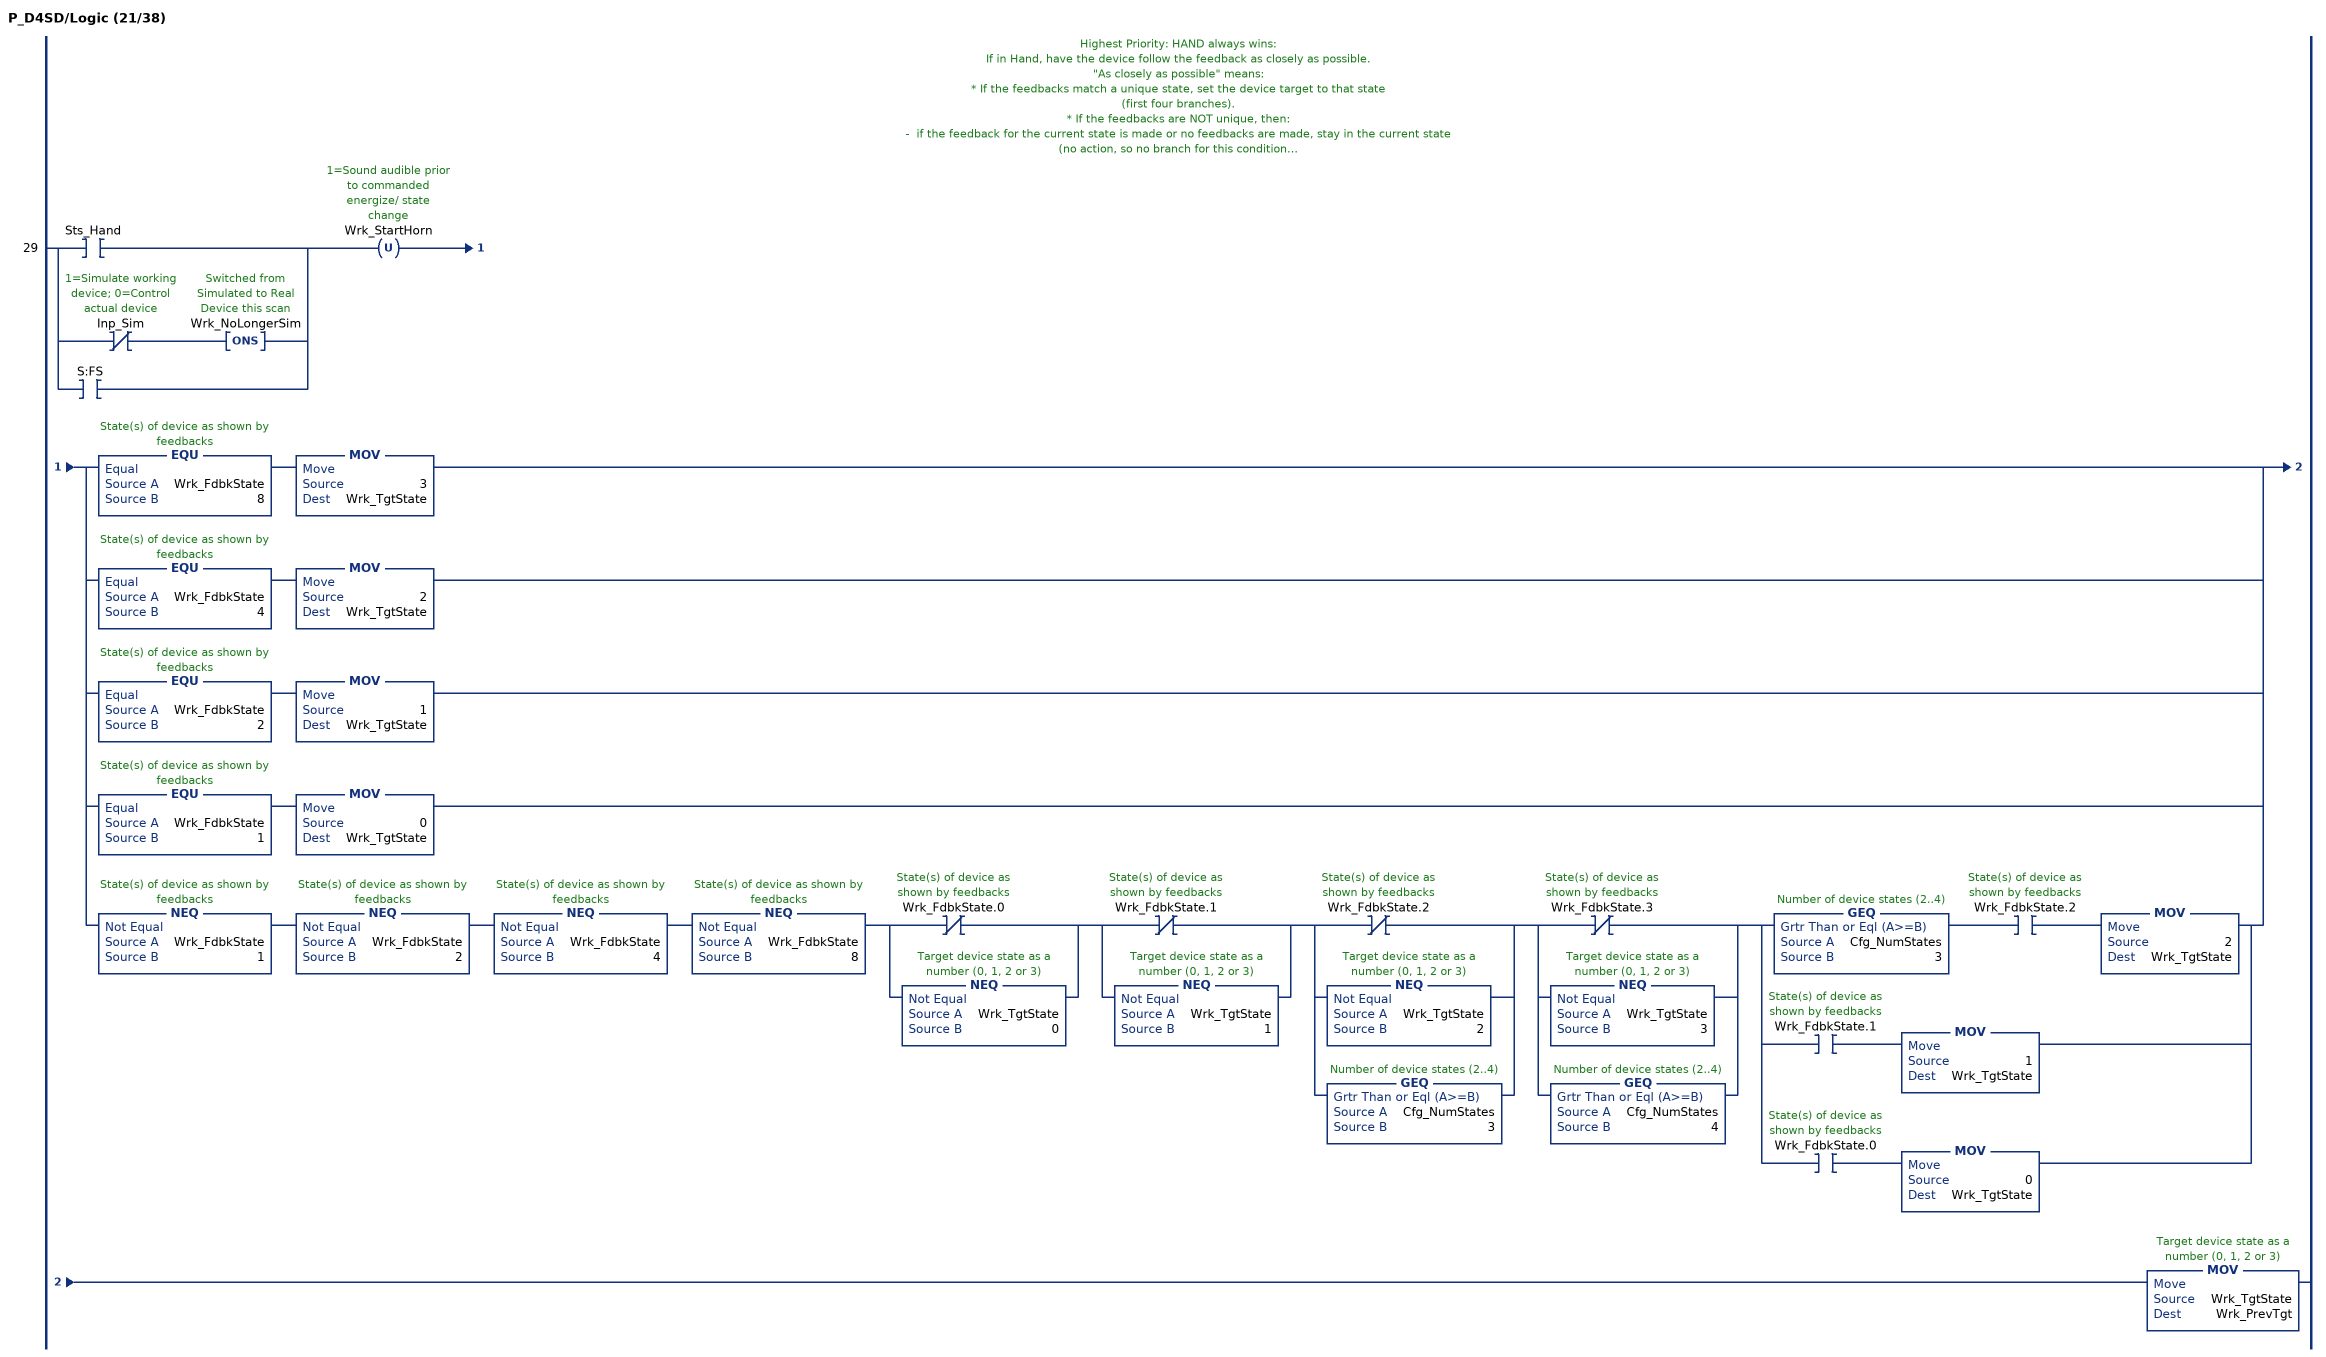
   // Highest Priority: HAND always wins:
   // If in Hand, have the device follow the feedback as closely as possible.
   // "As closely as possible" means:
   // * If the feedbacks match a unique state, set the device target to that state
   // (first four branches).
   // * If the feedbacks are NOT unique, then:
   // -  if the feedback for the current state is made or no feedbacks are made, stay in the current state
   // (no action, so no branch for this condition)
   // -  if multiple feedbacks are made but not the one for the current state, go to the lowest-numbered
   // state of the feedbacks that are made (bottom branch and its nested branches).
   // #####  V4.10.00  2019-03-08:  Added audible alert on commanded energize/state change.  #####
   29: [XIC(Sts_Hand) ,XIO(Inp_Sim) ONS(Wrk_NoLongerSim) ,XIC(S:FS) ]OTU(Wrk_StartHorn)[EQU(Wrk_FdbkState,8) MOV(3,Wrk_TgtState) ,EQU(Wrk_FdbkState,4) MOV(2,Wrk_TgtState) ,EQU(Wrk_FdbkState,2) MOV(1,Wrk_TgtState) ,EQU(Wrk_FdbkState,1) MOV(0,Wrk_TgtState) ,NEQ(Wrk_FdbkState,1) NEQ(Wrk_FdbkState,2) NEQ(Wrk_FdbkState,4) NEQ(Wrk_FdbkState,8) [XIO(Wrk_FdbkState.0) ,NEQ(Wrk_TgtState,0) ] [XIO(Wrk_FdbkState.1) ,NEQ(Wrk_TgtState,1) ] [XIO(Wrk_FdbkState.2) ,NEQ(Wrk_TgtState,2) ,GEQ(Cfg_NumStates,3) ] [XIO(Wrk_FdbkState.3) ,NEQ(Wrk_TgtState,3) ,GEQ(Cfg_NumStates,4) ] [GEQ(Cfg_NumStates,3) XIC(Wrk_FdbkState.2) MOV(2,Wrk_TgtState) ,XIC(Wrk_FdbkState.1) MOV(1,Wrk_TgtState) ,XIC(Wrk_FdbkState.0) MOV(0,Wrk_TgtState) ] ]MOV(Wrk_TgtState,Wrk_PrevTgt);
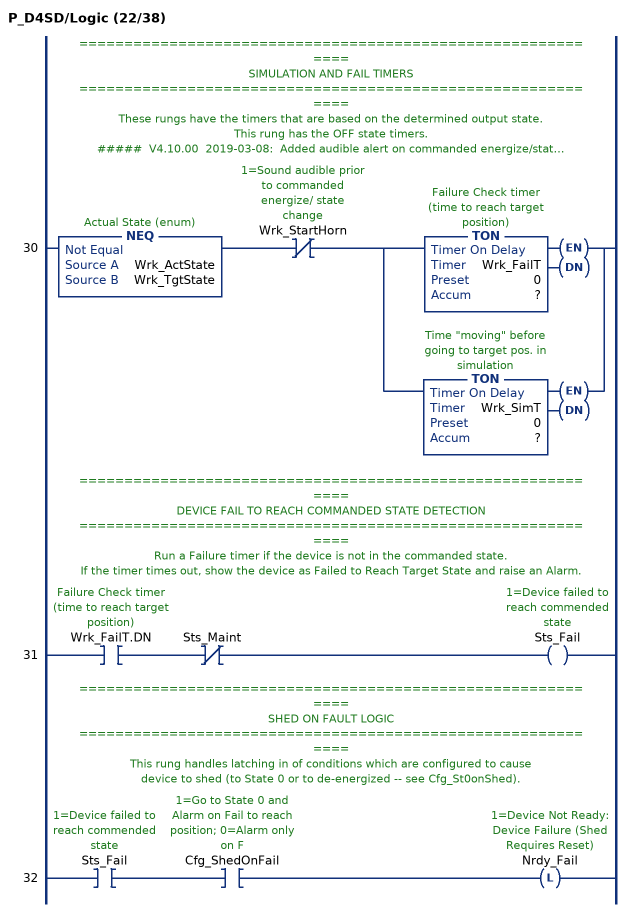
   // ============================================================
   // SIMULATION AND FAIL TIMERS
   // ============================================================
   // These rungs have the timers that are based on the determined output state.
   // This rung has the OFF state timers.
   // #####  V4.10.00  2019-03-08:  Added audible alert on commanded energize/state change.  #####
   30: NEQ(Wrk_ActState,Wrk_TgtState)XIO(Wrk_StartHorn)[TON(Wrk_FailT,?,?) ,TON(Wrk_SimT,?,?) ];
   // ============================================================
   // DEVICE FAIL TO REACH COMMANDED STATE DETECTION
   // ============================================================
   // Run a Failure timer if the device is not in the commanded state.
   // If the timer times out, show the device as Failed to Reach Target State and raise an Alarm.
   31: XIC(Wrk_FailT.DN)XIO(Sts_Maint)OTE(Sts_Fail);
   // ============================================================
   // SHED ON FAULT LOGIC
   // ============================================================
   // This rung handles latching in of conditions which are configured to cause
   // device to shed (to State 0 or to de-energized -- see Cfg_St0onShed).
   32: XIC(Sts_Fail)XIC(Cfg_ShedOnFail)OTL(Nrdy_Fail);
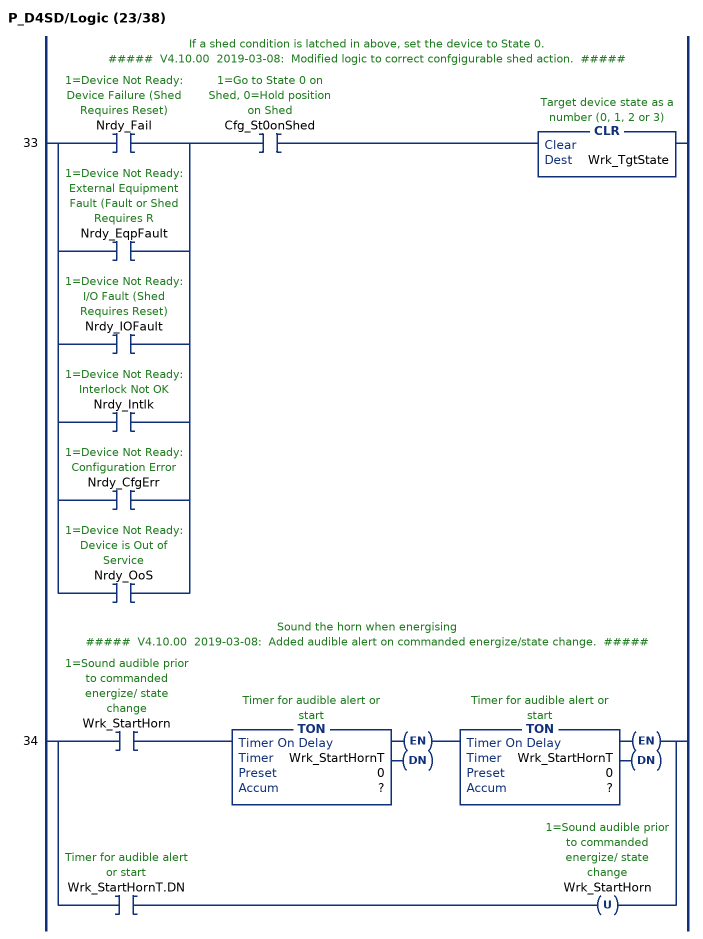
   // If a shed condition is latched in above, set the device to State 0.
   // #####  V4.10.00  2019-03-08:  Modified logic to correct confgigurable shed action.  #####
   33: [XIC(Nrdy_Fail) ,XIC(Nrdy_EqpFault) ,XIC(Nrdy_IOFault) ,XIC(Nrdy_Intlk) ,XIC(Nrdy_CfgErr) ,XIC(Nrdy_OoS) ]XIC(Cfg_St0onShed)CLR(Wrk_TgtState);
   // Sound the horn when energising
   // #####  V4.10.00  2019-03-08:  Added audible alert on commanded energize/state change.  #####
   34: [XIC(Wrk_StartHorn) TON(Wrk_StartHornT,?,?) TON(Wrk_StartHornT,?,?) ,XIC(Wrk_StartHornT.DN) OTU(Wrk_StartHorn) ];
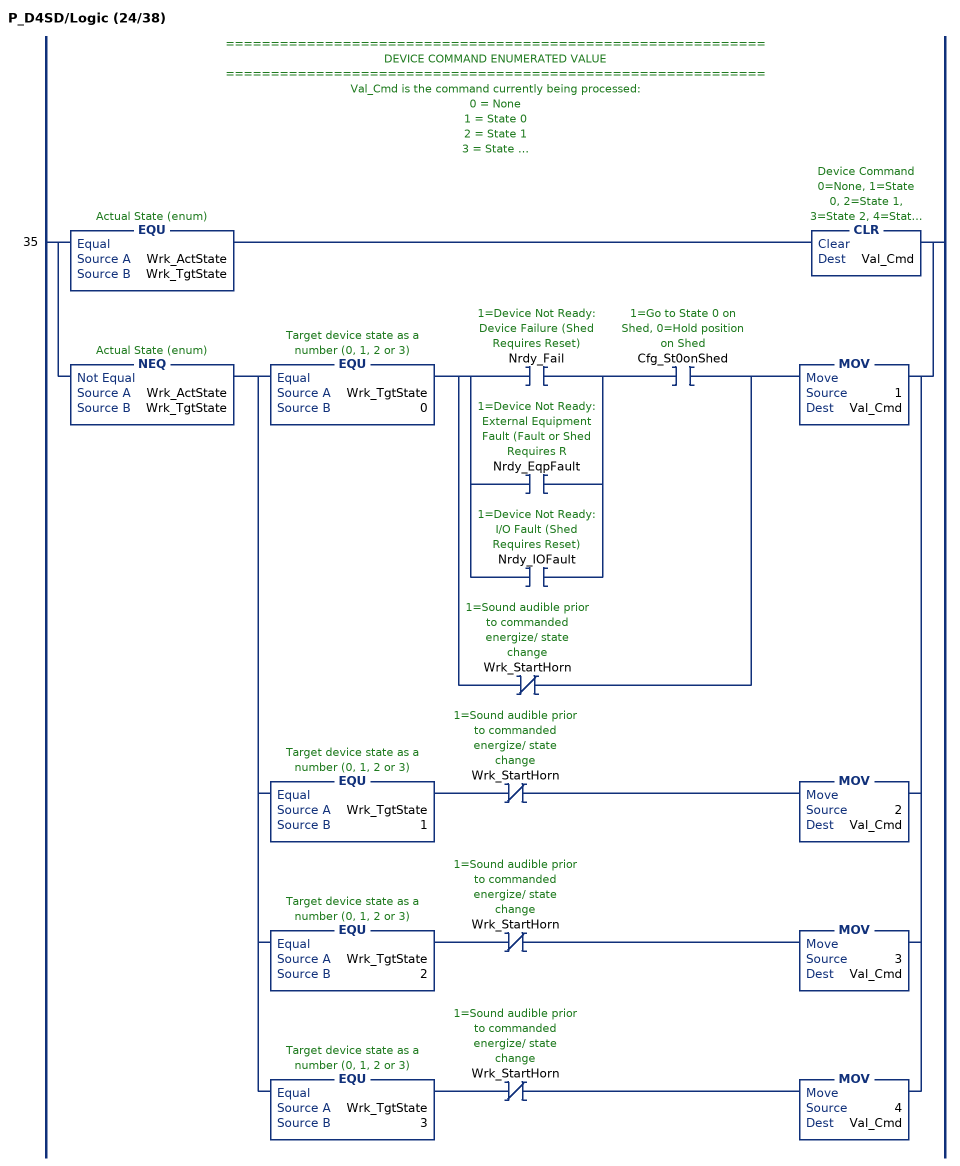
   // ============================================================
   // DEVICE COMMAND ENUMERATED VALUE
   // ============================================================
   // Val_Cmd is the command currently being processed:
   // 0 = None
   // 1 = State 0
   // 2 = State 1
   // 3 = State 2
   // 4 = State 3
   35: [EQU(Wrk_ActState,Wrk_TgtState) CLR(Val_Cmd) ,NEQ(Wrk_ActState,Wrk_TgtState) [EQU(Wrk_TgtState,0) [[XIC(Nrdy_Fail) ,XIC(Nrdy_EqpFault) ,XIC(Nrdy_IOFault) ] XIC(Cfg_St0onShed) ,XIO(Wrk_StartHorn) ] MOV(1,Val_Cmd) ,EQU(Wrk_TgtState,1) XIO(Wrk_StartHorn) MOV(2,Val_Cmd) ,EQU(Wrk_TgtState,2) XIO(Wrk_StartHorn) MOV(3,Val_Cmd) ,EQU(Wrk_TgtState,3) XIO(Wrk_StartHorn) MOV(4,Val_Cmd) ] ];
